# B&R Automation Studio project Parker_BMM_ST_V5_3147_V12 (part 30)

#### h_pid.c - Implementation code
```c
/********************************************************************
 * COPYRIGHT --
 ********************************************************************
 * Program: h_pid
 * File: h_pid.c
 * Author: lijianjun
 * Created: February 27, 2013
 ********************************************************************
 * Implementation of program h_pid -- heating and cooling controller
 ********************************************************************/

#include <bur/plctypes.h>
#include <string.h>

#ifdef _DEFAULT_INCLUDES
#include <AsDefault.h>
#endif

#include "edge.h"               /*edge function    */

#define  S$MODE_OFF					0
#define  S$MODE_PID					1
#define  S$MODE_TUNE					2

#define	C_STEP_WAIT 		   	0
#define	C_STEP_SYNC_HEAT_WAIT 	10
#define	C_STEP_HEAT 		    	20
#define	C_STEP_FREE 				30
#define	C_STEP_FREE_END			40
#define	C_STEP_COOL					50
#define	C_STEP_COOL_END 			60
#define	C_STEP_TUNE_END			70
#define	C_STEP_ERROR				999

void _INIT h_pidINIT(void)
{
	/* TODO: Add code here */
	gT_Par.Status.idxBroken = 0;
	gT_Par.Status.idxHigh   = 0;
	gT_Par.Status.idxLow    = 0;
	gT_Par.Status.idxFreeze = 0;
	gT_Par.Status.idxSwitchoff = 0;
	gT_Par.Status.idxNotNormal = 0;

	tProtectCooling = 0.0;

	/* ----- get task cycle time ----- */
	RTInfo_Task.enable = 1;
	RTInfo(&RTInfo_Task);

	tTask = RTInfo_Task.cycle_time/1000.0/1000.0;		/*  from us ---> s  */

	/* ----- setting tuning default value ----- */
	for(ZoneIndex=0; ZoneIndex<MAX_IDX_ZONE; ZoneIndex++)
	{
		/* parameter for tune   */
		LcrTempSet[ZoneIndex].TuneSet.delta_T_sync_heat = 40.0; 	 	/* Parameter for the synchronization  */
		LcrTempSet[ZoneIndex].TuneSet.delta_dT_sync_heat = 0.1;		/* Parameter for the synchronization d(temp)/dt  */
		LcrTempSet[ZoneIndex].TuneSet.cnt_wait_heat = 100;     		/* Parameter for the synchronization second  */

		LcrTempSet[ZoneIndex].TuneSet.delta_T_heat = 20.0;         	/* Parameter for the heating tuning 20 du */
		LcrTempSet[ZoneIndex].TuneSet.dT_min_heat  = 0.0;      		/* d(temp)/dt, min  */
		LcrTempSet[ZoneIndex].TuneSet.dRatio_heat  = 0.9;      		/* Internal parameter for the heating tuning 0 < dRatio_heat < 1*/
		LcrTempSet[ZoneIndex].TuneSet.cnt_tp_heat  = 180;      		/* 180  second */

		LcrTempSet[ZoneIndex].TuneSet.delta_T_sync_free  = 10.0; 	/* default value  */
		LcrTempSet[ZoneIndex].TuneSet.delta_dT_sync_free = 0.05;		/* default value   */
		LcrTempSet[ZoneIndex].TuneSet.cnt_wait_free      = 300;  	/* default value  300 second */

		LcrTempSet[ZoneIndex].TuneSet.delta_T_free = 10.0;				/* default value  10 du */
		LcrTempSet[ZoneIndex].TuneSet.dT_min_free  = 0.0;				/* default value  */
		LcrTempSet[ZoneIndex].TuneSet.dRatio_free  = 0.9;				/* default value  */
		LcrTempSet[ZoneIndex].TuneSet.cnt_tp_free  = 300;				/* default value  300 second */

		LcrTempSet[ZoneIndex].TuneSet.delta_T_sync_cool  = 10.0;		/* default value  10 du */
		LcrTempSet[ZoneIndex].TuneSet.delta_dT_sync_cool = 0.1;		/* not default value = 0.05  */
		LcrTempSet[ZoneIndex].TuneSet.cnt_wait_cool      = 300;		/* default value  300 second */

		LcrTempSet[ZoneIndex].TuneSet.delta_T_cool = 10.0;				/* default value  10 du */
		LcrTempSet[ZoneIndex].TuneSet.dT_min_cool  = 0.0;				/* default value  */
		LcrTempSet[ZoneIndex].TuneSet.dRatio_cool  = 0.9;				/* default value  */
		LcrTempSet[ZoneIndex].TuneSet.cnt_tp_cool  = 300.0;			/* default value  300 second */

		LcrTempSet[ZoneIndex].TuneSet.delta_T_sync_stop = 50.0;     /* Parameter for secure enable of the cooling tuning */
		LcrTempSet[ZoneIndex].TuneSet.filter_base_T = 20.0;         /* average value filter */
		LcrTempSet[ZoneIndex].TuneSet.Temp_amb = 40.0;

		LcrTempSet[ZoneIndex].TuneSet.mode = LCRTEMPTune_MODE_EXP;

		/* Heating and cooling mode  */
		LcrTempSet[ZoneIndex].enable_cooling  = 0;
		LcrTempSet[ZoneIndex].disable_heating = 0;

		/* stable parameter for PID   */
		LcrTempSet[ZoneIndex].PIDSet.hyst   = 2.0;
		LcrTempSet[ZoneIndex].PIDSet.Kw     = 1.0;
		LcrTempSet[ZoneIndex].PIDSet.delay  = 10.0;
		LcrTempSet[ZoneIndex].PIDSet.Kfbk   = 1.0;

		/* get address  */
		LCRTempTune_Array[ZoneIndex].pSettings = &(LcrTempSet[ZoneIndex]);
		LCRTempPID_Array[ZoneIndex].pSettings  = &(LcrTempSet[ZoneIndex]);

		gT_Par.Ctl.OnOff[ZoneIndex] = 0;
		gT_Par.Ctl.TuneOnOff[ZoneIndex] = 0;
		gT_Par.Ctl.IsHeatingOnPlan  = 0;
		gT_Par.Ctl.PreOnOff[ZoneIndex]= 0;
		gT_Par.Ctl.IsPreHeatingPlan = 0;

		OutBuffer[ZoneIndex]= 0.0;
		cntTask[ZoneIndex]  = 0;

		gT_Par.Status.TuneOk[ZoneIndex] = 0;

		HeatAlarm.tTempLow[ZoneIndex] = 1000.0;
	}/* for(ZoneIndex=0; ZoneIndex<MAX_ZoneIndex_CONTRL_ZONES; ZoneIndex++) */

}

void _CYCLIC h_pidCYCLIC(void)
{
	int i;
	gMachineInfo.bLoweringFlag =	bLowering; //ipis0424

	if (EDGEPOS(bLowering_Hmi,bLowering_Hmi_Pos))
	{
		if (1== gMachineOut.ParisonPump || 1== gMachineOut.ExtrA_Enable || 1==gMachineOut.ExtrB_Enable || gMachineOut.ExtrC_Enable || 1== gMachineOut.ExtrV_Enable)
		{
			gImply.ExtruderEnable =1;
		}
		else
		{
			bLowering =1;
		}
	}

	if (0==gMachineOut.HeatPower) //ipis0815
	{
		bLowering_Hmi =0;
	}

	if (0==bLowering_Hmi)
	{
		bLowering =0;
	}

	/* -------------------------------------------------------------------------- */
	if(1 == gT_Par.Ctl.IsAlarmConfirm)
	{
		gT_Par.Ctl.IsAlarmConfirm = 0;

		/* 非自复位的报警复位  */
		memset(gT_Par.Status.TempFreeze,0,sizeof(gT_Par.Status.TempFreeze));
		memset(gT_Par.Status.TempSwitchOff,0,sizeof(gT_Par.Status.TempSwitchOff));
	}

	/* -------------------------------------------------------------------------- */
	gT_Par.Status.idxBroken = 0;
	gT_Par.Status.idxHigh   = 0;
	gT_Par.Status.idxLow    = 0;
	gT_Par.Status.idxFreeze = 0;
	gT_Par.Status.idxSwitchoff = 0;
	gT_Par.Status.idxNotNormal = 0;

	gT_Par.Status.bBroken = 0;
	gT_Par.Status.bHigh   = 0;
	gT_Par.Status.bLowInternal = 0;
	gT_Par.Status.bFreeze = 0;
	gT_Par.Status.bSwitchOff = 0;
	gT_Par.Status.bNotNormal = 0;

	/*============================================================================*/
	/* Check group switches                              						         */
	/*============================================================================*/
	//	if(0 == gMachineIn.HeatingPowerNormal)gT_Par.GrpSwh.OnOff[0] = 0;
	if(0 == gMachineOut.HeatPower) gT_Par.GrpSwh.OnOff[0] = 0;

	if(0 == gT_Par.GrpSwh.OnOff[0] && 0 == gT_Par.GrpSwh.PreOnOff[0])
	{
		gMachineInfo.IsHeat = 0;
	}
	else if(1 == gT_Par.GrpSwh.OnOff[0] && 0 == gT_Par.GrpSwh.PreOnOff[0])
	{
		gMachineInfo.IsHeat = 1;
	}
	else
	{
		gMachineInfo.IsHeat = 2;
	}

	grpMaxIndex = sizeof(gT_Par.GrpSwh.OnOff)/sizeof(gT_Par.GrpSwh.OnOff[0]);
	if(grpMaxIndex > MAX_IDX_TEMPGROUP)grpMaxIndex = MAX_IDX_TEMPGROUP;

	for(grp=0; grp<grpMaxIndex; grp++)
	{
		if(gT_Par.Par.ST_GrpPreHeating[grp] < 20)gT_Par.Par.ST_GrpPreHeating[grp]= 20;
		if(gT_Par.Par.tGrpPreHeating[grp] < 10.0)gT_Par.Par.tGrpPreHeating[grp]  = 10.0;	/* 10.0min  */

		/* Pre-heating plan control  */
		if(1 == gT_Par.Ctl.IsPreHeatingPlan  && 0 == gT_Par.GrpSwh.PreOnOff[grp])
		{
			gMachineOut.HeatPower =1; //ipis0220
			gT_Par.GrpSwh.PreOnOff[grp] = 1;
			gT_Par.GrpSwh.OnOff[grp]    = 1;
		}

		if(1 == gT_Par.Ctl.IsHeatingOffPlan && 1 == gT_Par.GrpSwh.OnOff[grp])
		{
			gT_Par.GrpSwh.PreOnOff[grp] = 0;
		}

		if(0==gMachineIn.PreHeatDI)   //ipis0226
		{
			gT_Par.GrpSwh.PreOnOff[grp] = 0;
		}

		/* heating plan control  */
		if(1 == gT_Par.Ctl.IsHeatingOnPlan  && (0 == gT_Par.GrpSwh.OnOff[grp] || 1 == gT_Par.GrpSwh.PreOnOff[grp]))
		{
			gMachineOut.HeatPower =1; //ipis0220
			gT_Par.GrpSwh.OnOff[grp] = 1;
			gT_Par.GrpSwh.PreOnOff[grp] = 0;
		}

		if(1 == gT_Par.Ctl.IsHeatingOffPlan && 1 == gT_Par.GrpSwh.OnOff[grp])
		{
			gT_Par.GrpSwh.OnOff[grp] = 0;
		}

		/* Switch on group heating if group is on from VIS and programme enabled	*/
		if (EDGEPOS(gT_Par.GrpSwh.OnOff[grp],grp_OnOffPos[grp]))
		{
			HeatSequence[grp] = MAX_IDX_CONTRL_ZONES;
		}

		/* Switch off group heating if group is off from VIS and programe disabled	*/
		if (EDGENEG(gT_Par.GrpSwh.OnOff[grp],grp_OnOffNeg[grp]))
		{
			HeatSequence[grp] = 0;
			for(ZoneIndex=0;ZoneIndex<MAX_IDX_CONTRL_ZONES;ZoneIndex++)
			{
				if (gT_Par.Fix.SynchGroup[ZoneIndex] == grp)/*if grp nr configed     */
				{
					gT_Par.Ctl.OnOff[ZoneIndex] = 0;
				}
			}
		}
		/* Switch off group pre heating on  */
		if (EDGEPOS(gT_Par.GrpSwh.PreOnOff[grp],grp_PrePos[grp]))
		{
			for(ZoneIndex=0;ZoneIndex<MAX_IDX_CONTRL_ZONES;ZoneIndex++)
			{
				if (gT_Par.Fix.SynchGroup[ZoneIndex] == grp)/*if grp nr configed     */
				{
					gT_Par.Ctl.PreOnOff[ZoneIndex] = 1;
				}
			}
		}

		/* Switch off group pre heating off  */
		if (EDGENEG(gT_Par.GrpSwh.PreOnOff[grp],grp_PreNeg[grp]) || 0==gMachineIn.PreHeatDI) //ipis0221
		{
			for(ZoneIndex=0;ZoneIndex<MAX_IDX_CONTRL_ZONES;ZoneIndex++)
			{
				if (gT_Par.Fix.SynchGroup[ZoneIndex] == grp)/*if grp nr configed     */
				{
					gT_Par.Ctl.PreOnOff[ZoneIndex] = 0;
				}
			}
		}
		/* Switch off group tuning on  */
		if (EDGEPOS(gT_Par.GrpSwh.TuneOnOff[grp],grp_TunePos[grp]))
		{
			for(ZoneIndex=0;ZoneIndex<MAX_IDX_CONTRL_ZONES;ZoneIndex++)
			{
				if (gT_Par.Fix.SynchGroup[ZoneIndex] == grp)/*if grp nr configed     */
				{
					gT_Par.Ctl.TuneOnOff[ZoneIndex] = 1;
				}
			}
		}

		/* Switch off group tuning off  */
		if (EDGENEG(gT_Par.GrpSwh.TuneOnOff[grp],grp_TuneNeg[grp]))
		{
			for(ZoneIndex=0;ZoneIndex<MAX_IDX_CONTRL_ZONES;ZoneIndex++)
			{
				if (gT_Par.Fix.SynchGroup[ZoneIndex] == grp)/*if grp nr configed     */
				{
					gT_Par.Ctl.TuneOnOff[ZoneIndex] = 0;
				}
			}
		}

		grp_OnOffPos[grp] = gT_Par.GrpSwh.OnOff[grp];
		grp_OnOffNeg[grp] = gT_Par.GrpSwh.OnOff[grp];
	}/* for(grp=0; grp<grpMaxIndex; grp++) */

	/* Heat Sequence,one by one heat zone on */
	grpAct = grpMaxIndex;
	for(grp=0; grp<grpMaxIndex; grp++)
	{
		if(HeatSequence[grp] > 0)
		{
			grpAct = grp;
			break;
		}
	}

	if( grpAct < grpMaxIndex)
	{
		if(HeatSequence[grpAct] > 0)
		{
			if (grpAct == gT_Par.Fix.SynchGroup[MAX_IDX_CONTRL_ZONES - HeatSequence[grpAct]])
			{
				gT_Par.Ctl.OnOff[MAX_IDX_CONTRL_ZONES - HeatSequence[grpAct]] = 1;
			}
			HeatSequence[grpAct]--;
		}
	}

	/* check temperature change time  */
	if(gT_Par.Fix.tCheck < 10.0 )gT_Par.Fix.tCheck = 10.0;  /* 10.0s  */
	if(gT_Par.Fix.tHeatNormal < 20.0) gT_Par.Fix.tHeatNormal = 20.0;  /*  20.0 s */
	if(gT_Par.Fix.AT_MAX < 240.0)gT_Par.Fix.AT_MAX = 240.0; /* 240.0  */
	if(gT_Par.Par.ST_Tune_Same < 100)gT_Par.Par.ST_Tune_Same = 180.0;  /* Tune temperature   */

	/*============================================================================*/
	/* actual input && gAlarm check; PID parameters initialization   			  */
	/*============================================================================*/
	gMachineInfo.IsOpt = 0;
	for(ZoneIndex=0; ZoneIndex<MAX_IDX_CONTRL_ZONES; ZoneIndex++)
	{
		/*---UP-----------------------------------------------------------*/
		//		//		if (TempUpLimit_HMI[ZoneIndex]<=gT_Par.Fix.AT_MAX)
		//		//		{
		//		//			TempUpLimit_HMI[ZoneIndex] = gT_Par.Par.ST_PID[ZoneIndex]+  gUserFix_new.TempUpRange;
		//		//		}
		//		//		else
		//		//		{
		//		//			TempUpLimit_HMI[ZoneIndex] =gT_Par.Fix.AT_MAX;
		//		//		}
		//		//ipis022
		//		TempUpLimit_HMI[ZoneIndex] = gT_Par.Par.ST_PID[ZoneIndex]+  gUserFix_new.TempUpRange;
		//		if (gT_Par.Par.AlaUpTol[ZoneIndex] < gT_Par.Par.ST_PID[ZoneIndex] )
		//		{
		//			gT_Par.Par.AlaUpTol[ZoneIndex]=TempUpLimit_HMI[ZoneIndex];
		//		}
		//		//		if (gT_Par.Par.AlaUpTol[ZoneIndex] > gT_Par.Par.ST_PID[ZoneIndex] )
		//		//		{
		//		//			gT_Par.Par.AlaUpTol[ZoneIndex]=TempUpLimit_HMI[ZoneIndex];
		//		//		}
		//
		//		if (gT_Par.Par.AlaUpTol[ZoneIndex]>=TempUpLimit_HMI[ZoneIndex])
		//		{
		//			gT_Par.Par.AlaUpTol[ZoneIndex]=TempUpLimit_HMI[ZoneIndex];
		//		}
		//ipis0218
		if (gT_Par.Par.AlaUpTol[ZoneIndex] > gUserFix_new.TempUpRange )
		{
			gT_Par.Par.AlaUpTol[ZoneIndex]=gUserFix_new.TempUpRange;
		}
		if (gT_Par.Par.AlaUpTol[ZoneIndex] < 0 )
		{
			gT_Par.Par.AlaUpTol[ZoneIndex]=0;
		}
		/*---Down-----------------------------------------------------------*/
		//		if (TempUpLimit_HMI[ZoneIndex]>=0)
		//		{
		//			TempDwnLimit_HMI[ZoneIndex] = gT_Par.Par.ST_PID[ZoneIndex]- gUserFix_new.TempDwnRange;
		//		}
		//		else
		//		{
		//			TempDwnLimit_HMI[ZoneIndex] =0;
		//		}
		//		if(gT_Par.Par.AlaDwnTol[ZoneIndex]>gT_Par.Par.ST_PID[ZoneIndex])
		//		{
		//			gT_Par.Par.AlaDwnTol[ZoneIndex] = TempDwnLimit_HMI[ZoneIndex];
		//		}
		//		if(gT_Par.Par.AlaDwnTol[ZoneIndex]<TempDwnLimit_HMI[ZoneIndex])
		//		{
		//			gT_Par.Par.AlaDwnTol[ZoneIndex] = TempDwnLimit_HMI[ZoneIndex];
		//		}
		//
		//		if(gT_Par.Par.AlaDwnTol[ZoneIndex]<0)
		//		{
		//			gT_Par.Par.AlaDwnTol[ZoneIndex] = 0;
		//		}

		//ipis0218
		if(gT_Par.Par.AlaDwnTol[ZoneIndex]>gUserFix_new.TempDwnRange)
		{
			gT_Par.Par.AlaDwnTol[ZoneIndex] = gUserFix_new.TempDwnRange;
		}
		if(gT_Par.Par.AlaDwnTol[ZoneIndex]<0)
		{
			gT_Par.Par.AlaDwnTol[ZoneIndex] = 0;
		}

		/*---UP Same-----------------------------------------------------------*/
		//		if (TempUpLimit_Same_HMI<gT_Par.Fix.AT_MAX)
		//		{
		//			TempUpLimit_Same_HMI = gT_Par.Par.ST_PID_Same+  gUserFix_new.TempUpRange;
		//		}
		//		else
		//		{
		//			TempUpLimit_Same_HMI =gT_Par.Fix.AT_MAX;
		//		}
		//		TempUpLimit_Same_HMI = gT_Par.Par.ST_PID_Same+  gUserFix_new.TempUpRange;
		//		if (gT_Par.Par.AlaUpTol_Same<gT_Par.Par.ST_PID_Same)
		//		{
		//			gT_Par.Par.AlaUpTol_Same = TempUpLimit_Same_HMI;
		//		}
		//		//		if (gT_Par.Par.AlaUpTol_Same>gT_Par.Par.ST_PID_Same)
		//		//		{
		//		//			gT_Par.Par.AlaUpTol_Same = TempUpLimit_Same_HMI;
		//		//		}
		//		if (gT_Par.Par.AlaUpTol_Same>=TempUpLimit_Same_HMI)
		//		{
		//			gT_Par.Par.AlaUpTol_Same=TempUpLimit_Same_HMI;

		//ipis0218
		if (gT_Par.Par.AlaUpTol_Same > gUserFix_new.TempUpRange )
		{
			gT_Par.Par.AlaUpTol_Same=gUserFix_new.TempUpRange;
		}
		if (gT_Par.Par.AlaUpTol_Same < 0 )
		{
			gT_Par.Par.AlaUpTol_Same=0;
		}

		/*---Down Same-----------------------------------------------------------*/
		//		if (TempDwnLimit_Same_HMI>=0)
		//		{
		//			TempDwnLimit_Same_HMI = gT_Par.Par.ST_PID_Same- gUserFix_new.TempDwnRange;
		//		}
		//		else
		//		{
		//			TempDwnLimit_Same_HMI = 0;
		//		}
		//
		//		if (gT_Par.Par.AlaDwnTol_Same >gT_Par.Par.ST_PID_Same )
		//		{
		//			gT_Par.Par.AlaDwnTol_Same = TempDwnLimit_Same_HMI;
		//		}
		//		if (gT_Par.Par.AlaDwnTol_Same <TempDwnLimit_Same_HMI )
		//		{
		//			gT_Par.Par.AlaDwnTol_Same = TempDwnLimit_Same_HMI;
		//		}
		//		if (gT_Par.Par.AlaDwnTol_Same <0)
		//		{
		//			gT_Par.Par.AlaDwnTol_Same =0;
		//		}

		//ipis0218
		if(gT_Par.Par.AlaDwnTol_Same>gUserFix_new.TempDwnRange)
		{
			gT_Par.Par.AlaDwnTol_Same = gUserFix_new.TempDwnRange;
		}
		if(gT_Par.Par.AlaDwnTol_Same<0)
		{
			gT_Par.Par.AlaDwnTol_Same= 0;
		}

		//		TempUpLimit_HMI[ZoneIndex] = gT_Par.Par.ST_PID[ZoneIndex]+  gUserFix_new.TempUpRange;
		//
		//		TempDwnLimit_HMI[ZoneIndex] = gT_Par.Par.ST_PID[ZoneIndex]- gUserFix_new.TempDwnRange;
		//
		//		TempUpLimit_Same_HMI = gT_Par.Par.ST_PID_Same+  gUserFix_new.TempUpRange;
		//
		//		TempDwnLimit_Same_HMI = gT_Par.Par.ST_PID_Same- gUserFix_new.TempDwnRange;

		/*--------------------------------------------------------------*/

		gT_Par.Fix.bContactor[ZoneIndex] = 1;
		if(gT_Par.Fix.tTempFreeze[ZoneIndex] < 10.0 )gT_Par.Fix.tTempFreeze[ZoneIndex] = 10.0;
		if(gT_Par.Fix.tTempFreeze[ZoneIndex] > 1800.0)gT_Par.Fix.tTempFreeze[ZoneIndex] = 1800.0;

		if(tTask > 0.0 && 1 == gT_Par.Fix.Cooling[ZoneIndex])
		{
			gT_Par.Fix.tPeriodHeat[ZoneIndex] = ((INT)(gT_Par.Fix.tPeriodHeat[ZoneIndex]/tTask + 0.5)) * tTask;
			if(gT_Par.Fix.tPeriodHeat[ZoneIndex] < 10 * tTask)gT_Par.Fix.tPeriodHeat[ZoneIndex] = 10 * tTask;
		}

		if(tTask > 0.0 && 1 == gT_Par.Fix.bContactor[ZoneIndex])
		{
			gT_Par.Fix.tPeriodHeat[ZoneIndex] = ((INT)(gT_Par.Fix.tPeriodHeat[ZoneIndex]/tTask + 0.5)) * tTask;
			if(gT_Par.Fix.tPeriodHeat[ZoneIndex] < 10 * tTask)gT_Par.Fix.tPeriodHeat[ZoneIndex] = 10 * tTask;
		}

		/* ------ PID OPT value change ------ */
		if (memcmp(&gT_Par.Fix.ParTune[ZoneIndex],&ParTuneOld[ZoneIndex],sizeof(ParTuneOld[ZoneIndex])) != 0)
		{
			LcrTempSet[ZoneIndex].PIDpara = gT_Par.Fix.ParTune[ZoneIndex];
			LCRTempPID_Array[ZoneIndex].update = 1;
			ParTuneOld[ZoneIndex] = gT_Par.Fix.ParTune[ZoneIndex];
		}

		/* ---------------------- heating  normal -----------------------*/
		//ByPass gH_IO.HeatNormal(Feedback signal)which for detect heater error
		gH_IO.HeatNormal[ZoneIndex] = gH_IO.do_H[ZoneIndex];

		if(1 == gH_IO.do_H[ZoneIndex] && 0 == gH_IO.HeatNormal[ZoneIndex])
		{
			if(tHeatNormal[ZoneIndex] > 0.0)tHeatNormal[ZoneIndex] = tHeatNormal[ZoneIndex] - tTask;
			if(tHeatNormal[ZoneIndex] <= 0.0)
			{
				gT_Par.Status.bAlarmHeatNormal[ZoneIndex] = 1;
			}
		}
		else if(0 == gH_IO.do_H[ZoneIndex] && 1 == gH_IO.HeatNormal[ZoneIndex])
		{
			if(tHeatNormal[ZoneIndex] > 0.0)tHeatNormal[ZoneIndex] = tHeatNormal[ZoneIndex] - tTask;
			if(tHeatNormal[ZoneIndex] <= 0.0)
			{
				gT_Par.Status.bAlarmHeatNormal[ZoneIndex] = 1;
			}
		}
		else
		{
			gT_Par.Status.bAlarmHeatNormal[ZoneIndex] = 0;
			tHeatNormal[ZoneIndex] = gT_Par.Fix.tHeatNormal;
		}

		////ipis0719/////////////////////////////////////////////////////////////////////////////////////////////////////////////
		//		if (   0==TempInitOK[ZoneIndex]  )
		//		{
		//			//ipis0218
		//			if (( gH_IO.ActT[ZoneIndex] < gT_Par.Par.ST_PID[ZoneIndex] - gT_Par.Par.AlaDwnTol[ZoneIndex])&& 1 == gT_Par.Fix.Enable[ZoneIndex]
		//				|| 0==gMachineInfo.ExtrHeatTimeFlag) //ipis0213
		//			{
		//				gExtruderTempLow_HMIFlag =1;
		//			}
		//			else
		//			{
		//				gExtruderTempLow_HMIFlag =0;
		//			}
		//
		//		}

		/////////////////////////////////////////////////////////////////////////////////////////////////////////////////

		/* --- if current zone disabled, clear control bit --- */
		if (0 == gT_Par.Fix.Enable[ZoneIndex])
		{
			gT_Par.Ctl.OnOff[ZoneIndex] = 0;
			gT_Par.Ctl.TuneOnOff[ZoneIndex] = 0;

			gT_Par.Status.AlmHigh[ZoneIndex]      = 0;
			gT_Par.Status.AlmLow[ZoneIndex]       = 0;
			gT_Par.Status.SensorBroken[ZoneIndex] = 0;     /*For error bit show*/

			HeatAlarm.tSensorBroken[ZoneIndex] = 0.0;
			HeatAlarm.tTempHigh[ZoneIndex] = 0.0;
			HeatAlarm.tTempLow[ZoneIndex]  = 0.0;
			TempInitOK[ZoneIndex]=1;  //ipis0719

			//Bypass for gExtruderTempLow_HMIFlag
			TempProtection[ZoneIndex] =1;
			TempNotLow[ZoneIndex] =1;

		}
		else
		{
			if (1==gMachineInfo.IsHeat)
			{
				//	if (gH_IO.ActT[ZoneIndex] >= gT_Par.Par.AlaDwnTol[ZoneIndex])
				//ipis0218
				if (gH_IO.ActT[ZoneIndex] >= gT_Par.Par.ST_PID[ZoneIndex] - gT_Par.Par.AlaDwnTol[ZoneIndex])
				{
					{
						TempInitOK[ZoneIndex]=1;
					}

				}
				else
				{
					TempInitOK[ZoneIndex]=0;
				}

				if (1 == gT_Par.GrpSwh.OnOff[0])  //ipis 0128
				{
					gT_Par.Ctl.OnOff[ZoneIndex] = 1;
				}
				/*============================================================================*/
				/* Check gAlarm bit                                 						     */
				/*============================================================================*/
				/*-----------sensor broken or Opencircuit check-----------------------------*/
				if (gH_IO.ActT[ZoneIndex] >= 3000.0 || gH_IO.ActT[ZoneIndex] <= -3000.0)
				{
					HeatAlarm.tSensorBroken[ZoneIndex] = HeatAlarm.tSensorBroken[ZoneIndex] + tTask;

					if(HeatAlarm.tSensorBroken[ZoneIndex] > gT_Par.Fix.tCheck)
					{
						gT_Par.Status.SensorBroken[ZoneIndex] = 1;
					}
					else
					{
						gT_Par.Status.SensorBroken[ZoneIndex] = 0;
					}

					gT_Par.Status.AlmHigh[ZoneIndex] = 0;
					gT_Par.Status.AlmLow[ZoneIndex]  = 0;
					gT_Par.Status.TempFreeze[ZoneIndex] = 0;
				}
				else
				{
					HeatAlarm.tSensorBroken[ZoneIndex] = 0.0;
					gT_Par.Status.SensorBroken[ZoneIndex] = 0;

					if (1==gMachineInfo.IsHeat && (uDisHeaterTime>= gUserFix_new.HeatLowTimeOut*60))
					{
						//	if (gH_IO.ActT[ZoneIndex] < gT_Par.Par.AlaDwnTol[ZoneIndex])
						//ipis0218
						if (gH_IO.ActT[ZoneIndex] < gT_Par.Par.ST_PID[ZoneIndex]- gT_Par.Par.AlaDwnTol[ZoneIndex])
						{
							gAlarm.HeatError=1;
						}

					}

					if(1==TempInitOK[ZoneIndex] && 0== bLowering && 0==gT_Par.Ctl.IsPreHeatingPlan ) //ipis0304
					{
						/*Actual temperature high temp limit or upper tolerance limit*/
						//	if (gH_IO.ActT[ZoneIndex] > (gT_Par.Par.AlaUpTol[ZoneIndex]))/*Albert*/
						//ipis0211
						if (gH_IO.ActT[ZoneIndex] > (gT_Par.Par.ST_PID[ZoneIndex] +gT_Par.Par.AlaUpTol[ZoneIndex]))/*Albert*/
						{
							HeatAlarm.tTempHigh[ZoneIndex] = HeatAlarm.tTempHigh[ZoneIndex] + tTask;
							if(HeatAlarm.tTempHigh[ZoneIndex] > gT_Par.Fix.tCheck)
							{
								gT_Par.Status.AlmHigh[ZoneIndex] = 1;
							}
							else
							{
								gT_Par.Status.AlmHigh[ZoneIndex] = 0;
							}
						}
						else
						{
							HeatAlarm.tTempHigh[ZoneIndex] = 0.0;
							gT_Par.Status.AlmHigh[ZoneIndex] = 0;
						}

						/*Actual temperature low temp. limit or down tolerance limit*/
						//	if (gH_IO.ActT[ZoneIndex] < gT_Par.Par.AlaDwnTol[ZoneIndex])
						//ipis0218
						if (gH_IO.ActT[ZoneIndex] < gT_Par.Par.ST_PID[ZoneIndex] - gT_Par.Par.AlaDwnTol[ZoneIndex])

						{
							HeatAlarm.tTempLow[ZoneIndex] = HeatAlarm.tTempLow[ZoneIndex] + tTask;
							if(HeatAlarm.tTempLow[ZoneIndex] > gT_Par.Fix.tCheck)
							{
								gT_Par.Status.AlmLow[ZoneIndex] = 1;
							}
							else
							{
								gT_Par.Status.AlmLow[ZoneIndex] = 0;
							}
						}
						else
						{
							HeatAlarm.tTempLow[ZoneIndex] = 0.0;
							gT_Par.Status.AlmLow[ZoneIndex] = 0;
						}

						/*Actual temperature > permit max ---> stop heating */
						if ((gH_IO.ActT[ZoneIndex] > gT_Par.Fix.AT_MAX || gH_IO.ActT[ZoneIndex] < -100) &&
							(1 == gT_Par.Ctl.TuneOnOff[ZoneIndex] || 1 == gT_Par.Ctl.OnOff[ZoneIndex] || 1 == gT_Par.Ctl.PreOnOff[ZoneIndex])
							)
						{
							HeatAlarm.tTempSwitchOff[ZoneIndex] = HeatAlarm.tTempSwitchOff[ZoneIndex] + tTask;

							if(HeatAlarm.tTempSwitchOff[ZoneIndex] > gT_Par.Fix.tCheck)
							{
								gT_Par.Ctl.TuneOnOff[ZoneIndex] = 0;
								gT_Par.Ctl.OnOff[ZoneIndex]     = 0;
								gT_Par.Ctl.PreOnOff[ZoneIndex]  = 0;

								gT_Par.Status.TempSwitchOff[ZoneIndex] = 1;
							}
							else
							{
								gT_Par.Status.TempSwitchOff[ZoneIndex] = 0;
							}
						}
						else
						{
							HeatAlarm.tTempSwitchOff[ZoneIndex] = 0.0;
							gT_Par.Status.TempSwitchOff[ZoneIndex] = 0;

						}

					}
					else
					{
						gT_Par.Status.AlmHigh[ZoneIndex] = 0;
						gT_Par.Status.AlmLow[ZoneIndex] = 0;
						gT_Par.Status.TempSwitchOff[ZoneIndex] = 0;

					}

				}

			}

			//for gExtruderTempLow_HMIFlag
			if (gH_IO.ActT[ZoneIndex] > gUserFix_new.ProtectionTemp ) //ipis0225
			{
				TempProtection[ZoneIndex] =1;
			}
			else
			{
				TempProtection[ZoneIndex] =0;
			}

			if (gH_IO.ActT[ZoneIndex] < gT_Par.Par.ST_PID[ZoneIndex] - gT_Par.Par.AlaDwnTol[ZoneIndex] ) //0226
			{
				TempNotLow[ZoneIndex] =0;
			}
			else
			{
				TempNotLow[ZoneIndex] =1;
			}

		}/* if (0 == gT_Par.Fix.Enable[ZoneIndex]) */

		/* PID and TUNE get set parameter address  */
		LCRTempPID_Array[ZoneIndex].pSettings  = &LcrTempSet[ZoneIndex];
		LCRTempTune_Array[ZoneIndex].pSettings = &LcrTempSet[ZoneIndex];

		/* act temperature */
		LCRTempPID_Array[ZoneIndex].Temp  = gH_IO.ActT[ZoneIndex];
		LCRTempTune_Array[ZoneIndex].Temp = gH_IO.ActT[ZoneIndex];

		/*  set temperature */
		if(1 == gT_Par.Ctl.PreOnOff[ZoneIndex])
		{
			for(grp=0; grp<grpMaxIndex; grp++)
			{
				if (gT_Par.Fix.SynchGroup[ZoneIndex] == grp)
				{
					LCRTempPID_Array[ZoneIndex].Temp_set = gT_Par.Par.ST_GrpPreHeating[grp];
				}
			}
		}
		else
		{
			/*2018.7.31 Albert add new lowering setting*/
			//			LCRTempPID_Array[ZoneIndex].Temp_set = gT_Par.Par.ST_PID[ZoneIndex];
			if(1 == bLowering)	LCRTempPID_Array[ZoneIndex].Temp_set = gT_Par.Par.ST_PID[ZoneIndex] - gT_Par.Par.Lower;
			else LCRTempPID_Array[ZoneIndex].Temp_set = gT_Par.Par.ST_PID[ZoneIndex];

		}

		gT_Par.Par.ST_Tune[ZoneIndex] = gT_Par.Par.ST_Tune_Same;
		LCRTempTune_Array[ZoneIndex].Temp_set = gT_Par.Par.ST_Tune[ZoneIndex];

		//		/* Preheating on time --> Preheating off, normal heating*/
		//		if(1 == gT_Par.Ctl.PreOnOff[ZoneIndex])
		//		{
		//			/* reach setting pre-heating temperature - 5.0 */
		//			if( gH_IO.ActT[ZoneIndex] > LCRTempPID_Array[ZoneIndex].Temp_set - 5.0)
		//			{
		//				HeatTest.tPreHeating[ZoneIndex] = HeatTest.tPreHeating[ZoneIndex] + tTask;
		//			}
		//			else
		//			{
		//				HeatTest.tPreHeating[ZoneIndex] = 0.0;
		//			}
		//
		//			for(grp=0; grp<grpMaxIndex; grp++)
		//			{
		//				if (gT_Par.Fix.SynchGroup[ZoneIndex] == grp)
		//				{
		//					if(HeatTest.tPreHeating[ZoneIndex] > gT_Par.Par.tGrpPreHeating[grp] * 60)
		//					{
		//						gT_Par.Ctl.OnOff[ZoneIndex]    = 1;
		//						gT_Par.Ctl.PreOnOff[ZoneIndex] = 0;
		//						gT_Par.Status.PreHeatingOk[ZoneIndex] = 1;
		//					}
		//				}
		//			}
		//		}
		//		else
		//		{
		//			HeatTest.tPreHeating[ZoneIndex] = 0;
		//		}

		/* Heating Power not Normal, single zone not permit heating  */
		if(0 == gMachineIn.HeatingPowerNormal)
		{
			gT_Par.Ctl.OnOff[ZoneIndex] = 0;
			gT_Par.Ctl.PreOnOff[ZoneIndex] = 0;
		}

		/* off or PID or tuning  */
		if ((1 == gT_Par.Status.SensorBroken[ZoneIndex]) || (0 == gT_Par.Fix.Enable[ZoneIndex]))     /*sensor broken*/
		{
			PIDSTEP[ZoneIndex] = S$MODE_OFF;			/* If sensor error or not anble --> switch off zone		*/

			gT_Par.Ctl.OnOff[ZoneIndex]     = 0;
			gT_Par.Ctl.TuneOnOff[ZoneIndex] = 0;
			gT_Par.Ctl.PreOnOff[ZoneIndex]  = 0;

			gT_Par.Status.Tuning[ZoneIndex] = 0;
			gT_Par.Status.TuneStatus[ZoneIndex] = 0;
		}
		else if ((1 == gT_Par.Ctl.TuneOnOff[ZoneIndex]) && (1 == gT_Par.Ctl.OnOff[ZoneIndex]))
		{
			PIDSTEP[ZoneIndex] = S$MODE_TUNE;		/* Tune mode*/

			gT_Par.Status.Tuning[ZoneIndex] = 1;
			gMachineInfo.IsOpt  =  1;
		}
		else if ((1 == gT_Par.Ctl.OnOff[ZoneIndex]) || (1 == gT_Par.Ctl.PreOnOff[ZoneIndex]))
		{
			PIDSTEP[ZoneIndex] = S$MODE_PID;			/* PID mode*/

			gT_Par.Status.Tuning[ZoneIndex] = 0;
			gT_Par.Status.TuneStatus[ZoneIndex] = 0;
		}
		else
		{
			PIDSTEP[ZoneIndex] = S$MODE_OFF;

			gT_Par.Ctl.OnOff[ZoneIndex]     = 0;
			gT_Par.Status.Tuning[ZoneIndex] = 0;
		}

		/* step machine for temperature control  */
		switch (PIDSTEP[ZoneIndex])
		{
			case S$MODE_OFF:
					LcrTempSet[ZoneIndex].enable_cooling = 0;

				gH_IO.y_heat[ZoneIndex] = 0;
				gH_IO.y_cool[ZoneIndex] = 0;

				cntTask[ZoneIndex] = 0;
				OutBuffer[ZoneIndex] = 0.0;

				HeatTest.tTempFreeze[ZoneIndex] = 0.0;
				gT_Par.Status.PreHeatingOk[ZoneIndex] = 0;

				StepTune[ZoneIndex] = C_STEP_WAIT;

				LCRTempTune_Array[ZoneIndex].okToCool    = 0;
				LCRTempTune_Array[ZoneIndex].okToCoolEnd = 0;
				LCRTempTune_Array[ZoneIndex].okToFree    = 0;
				LCRTempTune_Array[ZoneIndex].okToFreeEnd = 0;
				LCRTempTune_Array[ZoneIndex].okToHeat    = 0;

				LCRTempPID_Array[ZoneIndex].enable  = 0;
				LCRTempTune_Array[ZoneIndex].enable = 0;

				gT_Par.Status.Out[ZoneIndex] = 0.0;
				break;

			case S$MODE_PID:
					LCRTempPID_Array[ZoneIndex].enable  = 1;
				LCRTempTune_Array[ZoneIndex].enable = 0;

				StepTune[ZoneIndex] = C_STEP_WAIT;

				LCRTempPID_Array[ZoneIndex].mode = LCRTEMPPID_MODE_AUTO;

				LcrTempSet[ZoneIndex].PIDpara = gT_Par.Fix.ParTune[ZoneIndex];

				/* heating default setting pid parameter  */
				if(0.0 == LcrTempSet[ZoneIndex].PIDpara.Kp_h)LcrTempSet[ZoneIndex].PIDpara.Kp_h = 3.0;
				if(0.0 == LcrTempSet[ZoneIndex].PIDpara.Tn_h)LcrTempSet[ZoneIndex].PIDpara.Tn_h = 5.0;
				if(0.0 == LcrTempSet[ZoneIndex].PIDpara.Tv_h)LcrTempSet[ZoneIndex].PIDpara.Tv_h = 1.0;

				/* ------ option cooling ------ */
				if(LcrTempSet[ZoneIndex].enable_cooling != gT_Par.Fix.Cooling[ZoneIndex])
				{
					LCRTempPID_Array[ZoneIndex].update = 1;
					LcrTempSet[ZoneIndex].enable_cooling = gT_Par.Fix.Cooling[ZoneIndex];
				}

				/* cooling default setting pid parameter  */
				if(LcrTempSet[ZoneIndex].PIDpara.Kp_c < 0.1)LcrTempSet[ZoneIndex].PIDpara.Kp_c = 6.0;
				LcrTempSet[ZoneIndex].PIDpara.Tn_c = 0.0;
				LcrTempSet[ZoneIndex].PIDpara.Tv_c = 0.0;
				if(0 == ZoneIndex)LcrTempSet[ZoneIndex].PIDpara.Kp_c = 5.0;
				/* Calling fuction LCRTempPID  */
				LCRTempPID(&LCRTempPID_Array[ZoneIndex]);

				if(0 == LcrTempSet[ZoneIndex].enable_cooling && 0 == gT_Par.Fix.bContactor[ZoneIndex])	/*  only heating && not contactor heating*/
				{
					gH_IO.y_heat[ZoneIndex] = LCRTempPID_Array[ZoneIndex].y_heat;
					gH_IO.y_cool[ZoneIndex] = LCRTempPID_Array[ZoneIndex].y_cool;
				}
				else   /* heating and cooling */
				{
					cntSamples[ZoneIndex] = (UINT)(gT_Par.Fix.tPeriodHeat[ZoneIndex]/tTask + 0.1);
					if(cntSamples[ZoneIndex] > 0)
					{
						if(0 == (cntTask[ZoneIndex] % cntSamples[ZoneIndex]))
						{
							OutBuffer[ZoneIndex] = OutBuffer[ZoneIndex] + (LCRTempPID_Array[ZoneIndex].y_heat - LCRTempPID_Array[ZoneIndex].y_cool)/cntSamples[ZoneIndex];
							if(OutBuffer[ZoneIndex] >= 100.0)
							{
								OutBuffer[ZoneIndex] = OutBuffer[ZoneIndex] - 100.0;
								gH_IO.y_heat[ZoneIndex] = 100.0;
								gH_IO.y_cool[ZoneIndex] = 0.0;
							}
							else if(OutBuffer[ZoneIndex] <= -100.0)
							{
								OutBuffer[ZoneIndex] = OutBuffer[ZoneIndex] + 100.0;
								gH_IO.y_heat[ZoneIndex] = 0.0;
								gH_IO.y_cool[ZoneIndex] = 100;
							}
							else
							{
								gH_IO.y_heat[ZoneIndex] = 0.0;
								gH_IO.y_cool[ZoneIndex] = 0.0;
							}
						}
						else
						{
							OutBuffer[ZoneIndex] = OutBuffer[ZoneIndex] + (LCRTempPID_Array[ZoneIndex].y_heat - LCRTempPID_Array[ZoneIndex].y_cool)/cntSamples[ZoneIndex];
						}
					}
					else
					{
						gH_IO.y_heat[ZoneIndex] = LCRTempPID_Array[ZoneIndex].y_heat;
						gH_IO.y_cool[ZoneIndex] = LCRTempPID_Array[ZoneIndex].y_cool;
					}
				}

				cntTask[ZoneIndex] = cntTask[ZoneIndex] ++;
				if(cntTask[ZoneIndex]>= 10000)cntTask[ZoneIndex]= 1000;

				/* zone output percent  */
				if(LCRTempPID_Array[ZoneIndex].y_heat > 0)
				{
					gT_Par.Status.Out[ZoneIndex] = LCRTempPID_Array[ZoneIndex].y_heat;
				}
				else if (LCRTempPID_Array[ZoneIndex].y_cool > 0)
				{
					gT_Par.Status.Out[ZoneIndex] = - LCRTempPID_Array[ZoneIndex].y_cool;
				}
				else
				{
					gT_Par.Status.Out[ZoneIndex] = 0.0;
				}

				/* Heating excption -- sensor   */
				if(100.0 == LCRTempPID_Array[ZoneIndex].y_heat)
				{
					HeatTest.tTempFreeze[ZoneIndex] = HeatTest.tTempFreeze[ZoneIndex] +  tTask;
				}
				else
				{
					HeatTest.tTempFreeze[ZoneIndex] = 0.0;
				}

				if(tTask * 2 == HeatTest.tTempFreeze[ZoneIndex])
				{
					HeatTest.LastTemp[ZoneIndex] = LCRTempPID_Array[ZoneIndex].Temp;
				}

				if(gT_Par.Fix.tTempFreeze[ZoneIndex] == HeatTest.tTempFreeze[ZoneIndex] + tTask * 2)
				{
					if(LCRTempPID_Array[ZoneIndex].Temp < HeatTest.LastTemp[ZoneIndex] + 1.0)
					{
						gT_Par.Status.TempFreeze[ZoneIndex] = 1;
						if(1 == gT_Par.Fix.ProtectEna[ZoneIndex])
						{
							gT_Par.Ctl.OnOff[ZoneIndex]    = 0;
							gT_Par.Ctl.PreOnOff[ZoneIndex] = 0;
						}
					}
				}
				break;

			case S$MODE_TUNE:
					LCRTempPID_Array[ZoneIndex].enable  = 0;
				LCRTempTune_Array[ZoneIndex].enable = 1;

				/* ------ option cooling ------ */
				if(LcrTempSet[ZoneIndex].enable_cooling != 0)
				{
					LCRTempPID_Array[ZoneIndex].update = 1;
					LcrTempSet[ZoneIndex].enable_cooling = 0;
				}

				cntTask[ZoneIndex] = 0;
				OutBuffer[ZoneIndex] = 0.0;

				/* tuning step machine   */
				switch (StepTune[ZoneIndex])
				{
					/* ------- step start ------- */
					case C_STEP_WAIT:
						if(1 == gT_Par.Ctl.TuneOnOff[ZoneIndex])
						{
							gT_Par.Status.TuneOk[ZoneIndex] = 0;
							LCRTempTune_Array[ZoneIndex].start = 1;
							StepTune[ZoneIndex] = C_STEP_SYNC_HEAT_WAIT;
						}
						break;

					/* ------- step sync heat ------- */
					case C_STEP_SYNC_HEAT_WAIT:

						LCRTempTune_Array[ZoneIndex].okToHeat = 1;

						for( i=0; i<MAX_IDX_CONTRL_ZONES;i++)
						{
							if(1 == gT_Par.Ctl.TuneOnOff[i])
							{
								gT_Par.Status.okToHeat[i] = LCRTempTune_Array[i].rdyToHeat;
							}
							else
							{
								gT_Par.Status.okToHeat[i] = 1;
							}

							LCRTempTune_Array[ZoneIndex].okToHeat = LCRTempTune_Array[ZoneIndex].okToHeat & gT_Par.Status.okToHeat[i];
						}

						if(1 == LCRTempTune_Array[ZoneIndex].okToHeat)
						{
							StepTune[ZoneIndex] = C_STEP_HEAT;
						}
						break;

					/* ------- step  heating ------- */
					case C_STEP_HEAT:

						LCRTempTune_Array[ZoneIndex].okToFree = 1;

						for( i=0; i<MAX_IDX_CONTRL_ZONES;i++)
						{
							if(1 == gT_Par.Ctl.TuneOnOff[i])
							{
								gT_Par.Status.okToFree[i] = LCRTempTune_Array[i].rdyToFree;
							}
							else
							{
								gT_Par.Status.okToFree[i] = 1;
							}

							LCRTempTune_Array[ZoneIndex].okToFree = LCRTempTune_Array[ZoneIndex].okToFree & gT_Par.Status.okToFree[i];
						}

						if(1 == LCRTempTune_Array[ZoneIndex].okToFree)
						{
							StepTune[ZoneIndex] = C_STEP_FREE;
						}
						break;

					/* ------- step  heating free ------- */
					case  C_STEP_FREE:

						LCRTempTune_Array[ZoneIndex].okToFreeEnd = 1;

						for( i=0; i<MAX_IDX_CONTRL_ZONES;i++)
						{
							if(1 == gT_Par.Ctl.TuneOnOff[i])
							{
								gT_Par.Status.okToFreeEnd[i] = LCRTempTune_Array[i].rdyToFreeEnd;
							}
							else
							{
								gT_Par.Status.okToFreeEnd[i] = 1;
							}

							LCRTempTune_Array[ZoneIndex].okToFreeEnd = LCRTempTune_Array[ZoneIndex].okToFreeEnd & gT_Par.Status.okToFreeEnd[i];
						}

						if(1 == LCRTempTune_Array[ZoneIndex].okToFreeEnd)
						{
							StepTune[ZoneIndex] = C_STEP_FREE_END;
						}
						break;

					/* ------- step  heating free end ------- */
					case C_STEP_FREE_END:

						LCRTempTune_Array[ZoneIndex].okToCool = 1;

						for( i=0; i<MAX_IDX_CONTRL_ZONES;i++)
						{
							if(1 == gT_Par.Ctl.TuneOnOff[i])
							{
								gT_Par.Status.okToCool[i] = LCRTempTune_Array[i].rdyToCool;
							}
							else
							{
								gT_Par.Status.okToCool[i] = 1;
							}

							LCRTempTune_Array[ZoneIndex].okToCool = LCRTempTune_Array[ZoneIndex].okToCool & gT_Par.Status.okToCool[i];
						}

						if(1 == LCRTempTune_Array[ZoneIndex].okToCool)
						{
							StepTune[ZoneIndex] = C_STEP_COOL;
						}
						break;
					/* ------- step  cooling ------- */
					case C_STEP_COOL:

						LCRTempTune_Array[ZoneIndex].okToCoolEnd = 1;

						for( i=0; i<MAX_IDX_CONTRL_ZONES;i++)
						{
							if(1 == gT_Par.Ctl.TuneOnOff[i])
							{
								gT_Par.Status.okToCoolEnd[i] = LCRTempTune_Array[i].rdyToCoolEnd;
							}
							else
							{
								gT_Par.Status.okToCoolEnd[i] = 1;
							}

							LCRTempTune_Array[ZoneIndex].okToCoolEnd = LCRTempTune_Array[ZoneIndex].okToCoolEnd & gT_Par.Status.okToCoolEnd[i];
						}

						if(1 == LCRTempTune_Array[ZoneIndex].okToCoolEnd)
						{
							StepTune[ZoneIndex] = C_STEP_COOL_END;
						}
						break;

					/* ------- step  cooling end ------- */
					case C_STEP_COOL_END:
						if(1 == LCRTempTune_Array[ZoneIndex].done)
						{
							gT_Par.Status.TuneOk[ZoneIndex] = 1;
							StepTune[ZoneIndex] = C_STEP_TUNE_END;
						}
						break;

					/* ------- step  tune end ------- */
					case C_STEP_TUNE_END:
						LCRTempTune_Array[ZoneIndex].start = 0;
						gT_Par.Ctl.TuneOnOff[ZoneIndex] = 0;

						gT_Par.Fix.ParTune[ZoneIndex] = LcrTempSet[ZoneIndex].PIDpara;

						StepTune[ZoneIndex] = C_STEP_WAIT;
						break;

					/* ------- step  heating error ------- */
					case C_STEP_ERROR:
						gT_Par.Ctl.TuneOnOff[ZoneIndex] = 0;
						gT_Par.Ctl.OnOff[ZoneIndex]     = 0;
						gT_Par.Ctl.PreOnOff[ZoneIndex]  = 0;
						break;

				}/* switch (StepTune[ZoneIndex]) */

				/* Calling fuction LCRTempTune  */
				LCRTempTune(&LCRTempTune_Array[ZoneIndex]);

				if(LCRTempTune_Array[ZoneIndex].status >= LCR_ERR_LCRPIDTune_ABORT && LCRTempTune_Array[ZoneIndex].status <= LCR_ERR_LCRPIDTune_W_CHANGED)
				{
					StepTune[ZoneIndex] = C_STEP_ERROR;
				}

				gT_Par.Status.TuneStatus[ZoneIndex] = StepTune[ZoneIndex];

				gH_IO.y_heat[ZoneIndex] = LCRTempTune_Array[ZoneIndex].y_heat;
				gH_IO.y_cool[ZoneIndex] = LCRTempTune_Array[ZoneIndex].y_cool;

				/* zone output percent  */
				if(LCRTempTune_Array[ZoneIndex].y_heat > 0)
				{
					gT_Par.Status.Out[ZoneIndex] = LCRTempTune_Array[ZoneIndex].y_heat;
				}
				else if (LCRTempTune_Array[ZoneIndex].y_cool > 0)
				{
					gT_Par.Status.Out[ZoneIndex] = - LCRTempTune_Array[ZoneIndex].y_cool;
				}
				else
				{
					gT_Par.Status.Out[ZoneIndex] = 0.0;
				}

				if(100.0 == LCRTempTune_Array[ZoneIndex].y_heat)
				{
					HeatTest.tTempFreeze[ZoneIndex] = HeatTest.tTempFreeze[ZoneIndex] +  tTask;
				}
				else
				{
					HeatTest.tTempFreeze[ZoneIndex] = 0.0;
				}

				if(tTask * 2 == HeatTest.tTempFreeze[ZoneIndex])
				{
					HeatTest.LastTemp[ZoneIndex] = LCRTempPID_Array[ZoneIndex].Temp;
				}

				if(gT_Par.Fix.tTempFreeze[ZoneIndex] == HeatTest.tTempFreeze[ZoneIndex] + tTask * 2)
				{
					if(LCRTempPID_Array[ZoneIndex].Temp < HeatTest.LastTemp[ZoneIndex] + 1.0)
					{
						gT_Par.Status.TempFreeze[ZoneIndex] = 1;
						if(1 == gT_Par.Fix.ProtectEna[ZoneIndex])
						{
							gT_Par.Ctl.OnOff[ZoneIndex] = 0;
						}
					}
				}
				break;
		}/* switch (PIDSTEP[ZoneIndex]) */

		/* ------------------ gAlarm idex information ------------------ */
		if(1 == gT_Par.Status.SensorBroken[ZoneIndex])
		{
			gT_Par.Status.idxBroken = ZoneIndex + 1;
			gT_Par.Status.bBroken = 1;
		}

		if(1 == gT_Par.Status.AlmHigh[ZoneIndex])
		{
			gT_Par.Status.idxHigh = ZoneIndex + 1;
			gT_Par.Status.bHigh = 1;
		}

		if(1 == gT_Par.Status.AlmLow[ZoneIndex])
		{
			gT_Par.Status.idxLow = ZoneIndex + 1;
			gT_Par.Status.bLowInternal = 1;
		}

		if(1 == gT_Par.Status.TempSwitchOff[ZoneIndex])
		{
			gT_Par.Status.idxSwitchoff = ZoneIndex + 1;
			gT_Par.Status.bSwitchOff = 1;
		}

		if(1 == gT_Par.Status.TempFreeze[ZoneIndex])
		{
			gT_Par.Status.idxFreeze = ZoneIndex + 1;
			gT_Par.Status.bFreeze = 1;
		}

		if(1 == gT_Par.Status.bAlarmHeatNormal[ZoneIndex])
		{
			gT_Par.Status.bNotNormal = 1;
			gT_Par.Status.idxNotNormal = ZoneIndex + 1;
		}

		TempInitOK_Old[ZoneIndex] =1; //ipis0218

	}/* for(ZoneIndex=0; ZoneIndex<MAX_ZoneIndex_CONTRL_ZONES; ZoneIndex++) */
	////ipis0218
	gTempfirstHeatOK = memcmp(&TempInitOK, &TempInitOK_Old , sizeof(TempInitOK));//0= all OK
	TempProtectionFlag = memcmp(&TempProtection, &TempInitOK_Old , sizeof(TempProtection));  //0= all OK
	TempNotLowFlag = memcmp(&TempNotLow, &TempInitOK_Old , sizeof(TempNotLow)); //0= all OK

	if (0==gMachineInfo.IsHeat)
	{
		TempProtectionFix_HMI =1;
	}
	if (EDGEPOS(gMachineInfo.IsHeat,IsHeatPos))
	{
		if (0==TempProtectionFlag)
		{
			TempProtectionMode =1; //mold
			TempProtectionFix_HMI =1;
		}
		else
		{
			TempProtectionMode =0;	//fix
			TempProtectionFix_HMI =0;
		}
	}

	//	if (0==gTempfirstHeatOK) //ipis0225
	if (1==gMachineInfo.IsHeat && 0==gTempfirstHeatOK)
	{
		if (0==TempProtectionMode) //fix ipis0225
		{
			//			if (tProtectCooling < gT_Par.Fix.tProtectCoolingFix+10)
			//			{
			//				tProtectCooling = tProtectCooling + tTask;
			//			}
			//			if (tProtectCooling > gT_Par.Fix.tProtectCoolingFix ) //ipis0218 force first power on and first heat, must wait 20min
			//			{
			//				gMachineInfo.ExtrHeatTimeFlag =1;
			//					TempProtectionFix_HMI =1;
			//			}
			if (tProtectCooling < gT_Par.Fix.tProtectCoolingFix+10 || tProtectCooling < gT_Par.Fix.tProtectCooling+10)
			{
				tProtectCooling = tProtectCooling + tTask;
				if(tProtectCooling > gT_Par.Fix.tProtectCoolingFix)
				{
					TempProtectionFix_HMI =1;
				}
			}
			if (tProtectCooling > gT_Par.Fix.tProtectCoolingFix  && tProtectCooling > gT_Par.Fix.tProtectCooling ) //ipis0218 force first power on and first heat, must wait 20min
			{
				gMachineInfo.ExtrHeatTimeFlag =1;
				TempProtectionFix_HMI =1;
			}
		}
		else
		{
			if (tProtectCooling < gT_Par.Fix.tProtectCooling+10)
			{
				tProtectCooling = tProtectCooling + tTask;
			}
			if (tProtectCooling > gT_Par.Fix.tProtectCooling )
			{
				gMachineInfo.ExtrHeatTimeFlag =1;
			}
		}
	}
	else
	{
		tProtectCooling =0;
		gMachineInfo.ExtrHeatTimeFlag =0;
	}

	//ipis0226
	//gTempfirstHeatOK  =
	// TempNotLowFlag = all enable zone temp is in setting range
	// gMachineInfo.ExtrHeatTimeFlag  =
	if (0==gTempfirstHeatOK && 0== TempNotLowFlag && 1==gMachineInfo.ExtrHeatTimeFlag) //ipis0213
	{
		gExtruderTempLow_HMIFlag =0;
	}
	else
	{
		gExtruderTempLow_HMIFlag =1;
	}

	//ipis0213 	/* extruder protection cooling   */
	//	if (0==gTempfirstHeatOK)
	//	{
	//		tProtectCooling = tProtectCooling + tTask;
	//
	//
	//		if (1== gMachineInfo.ExtrHeatTimeFlag) //=ipis0225
	//		{
	//			if (tProtectCooling < gT_Par.Fix.tProtectCooling+10)
	//			{
	//				tProtectCooling = tProtectCooling + tTask;
	//			}
	//		}
	//		else
	//		{
	//			if (tProtectCooling < gT_Par.Fix.tProtectCoolingFix+10)
	//			{
	//				tProtectCooling = tProtectCooling + tTask;
	//			}
	//		}
	//
	//
	//		if (1== gMachineInfo.ExtrHeatTimeFlag)
	//		{
	//			if (tProtectCooling > gT_Par.Fix.tProtectCooling )
	//			{
	//				gMachineInfo.ExtrHeatTimeFlag =1;
	//			}
	//		}
	//		else
	//		{
	//			if (tProtectCooling > gT_Par.Fix.tProtectCoolingFix ) //ipis0218 force first power on and first heat, must wait 20min
	//			{
	//				gMachineInfo.ExtrHeatTimeFlag =1;
	//			}
	//
	//		}
	//
	//	}
	//	else
	//	{
	//		tProtectCooling =0;
	//		gMachineInfo.ExtrHeatTimeFlag =0;
	//	}

	/* extruder protection cooling   */
	if(0 == gT_Par.Status.bLowInternal)
	{
		//		tProtectCooling = tProtectCooling + tTask;
		//		if(tProtectCooling > 2 * gT_Par.Fix.tProtectCooling)
		//		{
		//			tProtectCooling = 2 * gT_Par.Fix.tProtectCooling + 1.0;
		//		}
		gT_Par.Status.bLow = 0;
		//		if(tProtectCooling >= gT_Par.Fix.tProtectCooling)
		//		{
		//			gT_Par.Status.bLow = 0;
		//		}
		//		else
		//		{
		//			gT_Par.Status.bLow = 1;
		//		}
	}
	else
	{
		//		tProtectCooling = 0.0;
		gT_Par.Status.bLow = 1;
		//	gT_Par.Status.bLow = 0; //ipis0227
	}

	/*2018.7.24 Albert add timer show heat time*/
	if(gMachineInfo.IsHeat && 0== bLowering)
	{
		rHeaterTime += tTask;
	}
	else
	{
		rHeaterTime = 0;
	}
	uDisHeaterTime = rHeaterTime;

}/* end of CYCLIC   */
```

#### h_pid.typ - Local data types
```iecst
(********************************************************************
 * COPYRIGHT --
 ********************************************************************
 * Program: h_pid
 * File: h_pid.typ
 * Author: lij
 * Created: February 27, 2013
 ********************************************************************
 * Local data types of program h_pid
 ********************************************************************)

TYPE
	Heat_Alarm_typ : 	STRUCT
		tTempSwitchOff : ARRAY[0..MAX_IDX_ZONE]OF REAL;
		tSensorBroken : ARRAY[0..MAX_IDX_ZONE]OF REAL;
		tTempHigh : ARRAY[0..MAX_IDX_ZONE]OF REAL;
		tTempLow : ARRAY[0..MAX_IDX_ZONE]OF REAL;
	END_STRUCT;
	Heat_Test_typ : 	STRUCT
		LastTemp : ARRAY[0..MAX_IDX_ZONE]OF REAL;
		tTempFreeze : ARRAY[0..MAX_IDX_ZONE]OF REAL;
		tPreHeating : ARRAY[0..MAX_IDX_ZONE]OF REAL;
	END_STRUCT;
END_TYPE
```

#### h_pid.var - Local variables
```iecst
(********************************************************************
 * COPYRIGHT --
 ********************************************************************
 * Program: h_pid
 * File: h_pid.var
 * Author: lij
 * Created: February 27, 2013
 ********************************************************************
 * Local variables of program h_pid
 ********************************************************************)
VAR
	ZoneIndex : UINT;
	tTask : REAL := 0.0;
	tProtectCooling : REAL;
	StepTune : ARRAY[0..MAX_IDX_ZONE] OF UINT;
	RTInfo_Task : RTInfo := (0);
	PIDSTEP : ARRAY[0..MAX_IDX_ZONE] OF UINT;
	ParTuneOld : ARRAY[0..MAX_IDX_ZONE] OF lcrtemp_pid_opt_typ;
	LCRTempTune_Array : ARRAY[0..MAX_IDX_ZONE] OF LCRTempTune := [MAX_IDX_ZONE+1(0)];
END_VAR
VAR RETAIN
	LcrTempSet : ARRAY[0..MAX_IDX_ZONE] OF lcrtemp_set_typ;
END_VAR
VAR
	LCRTempPID_Array : ARRAY[0..MAX_IDX_ZONE] OF LCRTempPID := [MAX_IDX_ZONE+1(0)];
	tHeatNormal : ARRAY[0..MAX_IDX_ZONE] OF REAL;
	OutBuffer : ARRAY[0..MAX_IDX_ZONE] OF REAL;
	cntTask : ARRAY[0..MAX_IDX_ZONE] OF UDINT;
	cntSamples : ARRAY[0..MAX_IDX_ZONE] OF UINT;
	HeatTest : Heat_Test_typ := (0);
	HeatSequence : ARRAY[0..MAX_IDX_TEMPGROUP] OF UINT := [MAX_IDX_TEMPGROUP+1(0)];
	HeatAlarm : Heat_Alarm_typ := (0);
	grp_TunePos : ARRAY[0..MAX_IDX_TEMPGROUP] OF BOOL;
	grp_TuneNeg : ARRAY[0..MAX_IDX_TEMPGROUP] OF BOOL;
	grp_PrePos : ARRAY[0..MAX_IDX_TEMPGROUP] OF BOOL;
	grp_PreNeg : ARRAY[0..MAX_IDX_TEMPGROUP] OF BOOL;
	grp_OnOffPos : ARRAY[0..MAX_IDX_TEMPGROUP] OF BOOL;
	grp_OnOffNeg : ARRAY[0..MAX_IDX_TEMPGROUP] OF BOOL;
	grpAct : UINT := 0;
	grpMaxIndex : UINT;
	grp : UINT := 0;
END_VAR
(*Heat  show Time*)
VAR
	uDisHeaterTime : UDINT;
	rHeaterTime : REAL;
END_VAR
(*Lowering Option*)
VAR
	bLowering : BOOL;
	TempUpLimit_HMI : ARRAY[0..MAX_IDX_ZONE] OF REAL;
	TempDwnLimit_HMI : ARRAY[0..MAX_IDX_ZONE] OF REAL;
	TempUpLimit_Same_HMI : REAL;
	TempDwnLimit_Same_HMI : REAL;
	TempInitOK : ARRAY[0..MAX_IDX_ZONE] OF REAL;
	bLowering_Hmi : BOOL;
	bLowering_Hmi_Pos : BOOL;
	TempInitOK_Old : ARRAY[0..MAX_IDX_ZONE] OF REAL;
	TempProtection : ARRAY[0..MAX_IDX_ZONE] OF REAL;
	TempProtectionFlag : BOOL;
	IsHeatPos : BOOL;
	TempProtectionMode : BOOL;
	TempProtectionFix_HMI : USINT;
	TempNotLow : ARRAY[0..MAX_IDX_ZONE] OF REAL;
	TempNotLowFlag : BOOL;
END_VAR
```

- edge.h (reference to Logical/GlobalIncludes/edge.h)

### Program Logical/Heating/h_pwm (ANSIC, version 1.00.0) - heating and cooling PWM

#### h_pwm.c - Implementation code
```c
/********************************************************************
 * COPYRIGHT --
 ********************************************************************
 * Program: h_pwm
 * File: h_pwm.c
 * Author: lijianjun
 * Created: March 04, 2013
 ********************************************************************
 * Implementation of program h_pwm --- heating and cooling PWM mode
 ********************************************************************/

#include <bur/plctypes.h>

#ifdef _DEFAULT_INCLUDES
	#include <AsDefault.h>
#endif

void _INIT h_pwmINIT(void)
{
	/* TODO: Add code here */
	gT_Par.GrpSwh.OnOff[0] = 0;
	for(ZoneIndex=0; ZoneIndex<MAX_IDX_CONTRL_ZONES; ZoneIndex++)
	{
		gT_Par.Ctl.OnOff[ZoneIndex] = 0;

		/* Heating time minum and Period  */
		gT_Par.Fix.tMinHeat[ZoneIndex]    = 0.05;
		gT_Par.Fix.tPeriodHeat[ZoneIndex] = 3.0;

        /* Cooling time minum and Period  */
		gT_Par.Fix.tMinCool[ZoneIndex]    = 0.2;
		gT_Par.Fix.tPeriodCool[ZoneIndex] = 3.0;

		LCRPWM_HeatArray[ZoneIndex].max_value = 100.0;
		LCRPWM_HeatArray[ZoneIndex].min_value = 0.0;

		LCRPWM_CoolArray[ZoneIndex].max_value = 100.0;
		LCRPWM_CoolArray[ZoneIndex].min_value = 0.0;
	}/* for(ZoneIndex=0; ZoneIndex<MAX_IDX_CONTRL_ZONES; ZoneIndex++) */
}

void _CYCLIC h_pwmCYCLIC(void)
{
	/* TODO: Add code here */

		/* quick setting parameters  */
		if(1 == gT_Par.Ctl.IsQuickSetValue && 0 == IsQuickSetValueOld)
		{
			gT_Par.Ctl.IsQuickSetValue = 0;
			for(ZoneIndex=0; ZoneIndex<MAX_IDX_ZONE; ZoneIndex++)
			{
				if(gT_Par.Par.ST_PID_Same > 0&& gT_Par.Par.ST_PID_Same <=gT_Par.Fix.AT_MAX)
				{
					gT_Par.Par.ST_PID[ZoneIndex] = gT_Par.Par.ST_PID_Same;
				}

				if(gT_Par.Par.AlaUpTol_Same > 0&& gT_Par.Par.AlaUpTol_Same <=gUserFix_new.TempUpRange)
				{
					gT_Par.Par.AlaUpTol[ZoneIndex] = gT_Par.Par.AlaUpTol_Same;
				}

				if(gT_Par.Par.AlaDwnTol_Same > 0&& gT_Par.Par.AlaDwnTol_Same <=gUserFix_new.TempDwnRange)
				{
					gT_Par.Par.AlaDwnTol[ZoneIndex] = gT_Par.Par.AlaDwnTol_Same;
				}
			}
		}/* if(1 == gT_Par.Ctl.IsQuickSetValue && 0 == IsQuickSetValueOld) */

		IsQuickSetValueOld = gT_Par.Ctl.IsQuickSetValue;

		bHeating = 0;
		for(ZoneIndex=0; ZoneIndex<MAX_IDX_CONTRL_ZONES; ZoneIndex++)
		{
			if(1 == gT_Par.Ctl.PreOnOff[ZoneIndex] || gT_Par.Ctl.OnOff[ZoneIndex])bHeating = 1;

			/* default heating pwm parameter */
			if(gT_Par.Fix.tMinHeat[ZoneIndex] < 0.05  )gT_Par.Fix.tMinHeat[ZoneIndex] = 0.05;
			if(1 == gT_Par.Fix.bContactor[ZoneIndex] && gT_Par.Fix.tMinHeat[ZoneIndex] < 0.3)gT_Par.Fix.tMinHeat[ZoneIndex] = 0.3;

			LCRPWM_HeatArray[ZoneIndex].enable = gT_Par.Fix.Enable[ZoneIndex];
			LCRPWM_HeatArray[ZoneIndex].t_min_pulse = gT_Par.Fix.tMinHeat[ZoneIndex];
			LCRPWM_HeatArray[ZoneIndex].t_period = gT_Par.Fix.tPeriodHeat[ZoneIndex];
			LCRPWM_HeatArray[ZoneIndex].x = gH_IO.y_heat[ZoneIndex];
			LCRPWM(&LCRPWM_HeatArray[ZoneIndex]);

			/* default cooling pwm parameter */
			if(gT_Par.Fix.tMinCool[ZoneIndex] < 0.3)gT_Par.Fix.tMinCool[ZoneIndex] = 0.3;
			gT_Par.Fix.tPeriodCool[ZoneIndex] = gT_Par.Fix.tPeriodHeat[ZoneIndex];

			LCRPWM_CoolArray[ZoneIndex].enable = gT_Par.Fix.Cooling[ZoneIndex];
			LCRPWM_CoolArray[ZoneIndex].t_min_pulse = gT_Par.Fix.tMinCool[ZoneIndex];
			LCRPWM_CoolArray[ZoneIndex].t_period = gT_Par.Fix.tPeriodCool[ZoneIndex];
			LCRPWM_CoolArray[ZoneIndex].x = gH_IO.y_cool[ZoneIndex];
			LCRPWM(&LCRPWM_CoolArray[ZoneIndex]);

			/* digital output  */
			gH_IO.do_H[ZoneIndex] = LCRPWM_HeatArray[ZoneIndex].pulse;
			gH_IO.do_C[ZoneIndex] = LCRPWM_CoolArray[ZoneIndex].pulse;

			/* analog output  */
			gH_IO.ao_H[ZoneIndex] = (INT)(gH_IO.y_heat[ZoneIndex] * 32767/100.0);
			gH_IO.ao_C[ZoneIndex] = (INT)(gH_IO.y_cool[ZoneIndex] * 32767/100.0);

			/* zones color  */

			if(1 == gT_Par.Status.SensorBroken[ZoneIndex])
			{
				gH_IO.ZoneColor[ZoneIndex] = 0x332A;	/* 红字黄底  *//*Word Red , Back Color Yellow*/
			}
			else if(1 == gT_Par.Status.AlmHigh[ZoneIndex])
			{
				gH_IO.ZoneColor[ZoneIndex] = 0x0137;   /* 蓝字红底  */	//*Word Blue , Back Color Red*/
			}
			else if(1 == gT_Par.Status.AlmLow[ZoneIndex])
			{
				gH_IO.ZoneColor[ZoneIndex] = 0x0110;	/* 蓝字白底  */	//*Word Blue , Back Color White*/
			}
			else
			{
				gH_IO.ZoneColor[ZoneIndex] = 0x0122;   /* 藍字黃底  */	//*Word Blue , Back Color Yellow*/
			}

			if(1 == gT_Par.Ctl.PreOnOff[ZoneIndex] )  /* 保温过程   */
			{
				gH_IO.ZoneColor[ZoneIndex] = 0x012F;   /* 蓝字黄底  */  //*Word Blue , Back Color Yellow*/
			}
			/***************************************************************************/
			/********************温区状态图组中的图片控制*******************************/
			/***************************************************************************/
			TON_StatusBG[ZoneIndex].IN = 1;

			if ((1 == gH_IO.do_H[ZoneIndex]) && (gH_IO.HC_sta[ZoneIndex] > 4))
			{
				gH_IO.HC_sta[ZoneIndex] = 4;
			}
			else if ((1 == gH_IO.do_C[ZoneIndex]) && (gH_IO.HC_sta[ZoneIndex] < 5))
			{
				gH_IO.HC_sta[ZoneIndex] = 5;
			}

			if (TON_StatusBG[ZoneIndex].Q == 1) 		/* 每1秒钟, 刷新图片 */
			{
				TON_StatusBG[ZoneIndex].IN = 0;

				if (1 ==gT_Par.Status.SensorBroken[ZoneIndex])
				{
					gH_IO.HC_sta[ZoneIndex] = 7;
				}
				else if (1 == gH_IO.do_H[ZoneIndex])
				{
					gH_IO.HC_sta[ZoneIndex] = gH_IO.HC_sta[ZoneIndex] + 1;

					if (gH_IO.HC_sta[ZoneIndex] > 4)
					{
						gH_IO.HC_sta[ZoneIndex] = 1;
					}
				}
				else if (1 == gH_IO.do_C[ZoneIndex])
				{
					gH_IO.HC_sta[ZoneIndex] = gH_IO.HC_sta[ZoneIndex] + 1;

					if (gH_IO.HC_sta[ZoneIndex] > 6)
					{
						gH_IO.HC_sta[ZoneIndex] = 5;
					}
				}
				else
				{
					gH_IO.HC_sta[ZoneIndex] = 0;
				}
			}/* if (TON_StatusBG[ZoneIndex].Q == 1) */

			/*********************************************************************************/
			/**************TON_StatusBG定时器实现*********************************************/
			/*********************************************************************************/
			TON_StatusBG[ZoneIndex].PT = 1000;				/*设定时间为1秒*/
			TON(&TON_StatusBG[ZoneIndex]);
		}/* for(ZoneIndex=0; ZoneIndex<MAX_IDX_CONTRL_ZONES; ZoneIndex++) */

		/* -------- 超溫保護開關 -------- */
		if(1 == gT_Par.Status.bSwitchOff)
		{
			gMachineOut.TempProtection = 1;
		}
		else
		{
			gMachineOut.TempProtection = 0;
		}
	}/* end of cyclic  */

void _EXIT h_pwmEXIT(void)
{
	/* TODO: Add code here */
}
```

#### h_pwm.var - Local variables
```iecst
(********************************************************************
 * COPYRIGHT --
 ********************************************************************
 * Program: h_pwm
 * File: h_pwm.var
 * Author: lij
 * Created: March 04, 2013
 ********************************************************************
 * Local variables of program h_pwm
 ********************************************************************)
VAR
	IsQuickSetValueOld : BOOL;
	bHeating : BOOL;
	ZoneIndex : UINT := 0;
	TON_StatusBG : ARRAY[0..MAX_IDX_ZONE] OF TON;
	LCRPWM_HeatArray : ARRAY[0..MAX_IDX_ZONE] OF LCRPWM := [MAX_IDX_ZONE+1(0)];
	LCRPWM_CoolArray : ARRAY[0..MAX_IDX_ZONE] OF LCRPWM := [MAX_IDX_ZONE+1(0)];
END_VAR
```

### Program Logical/Heating/trend (ANSIC, version 1.00.0) - temperature trend

#### trend.typ - Local data types
```iecst
(********************************************************************
 * COPYRIGHT --  B&R
 ********************************************************************
 * Program: trend
 * File: trend.typ
 * Author: lij
 * Created: March 06, 2013
 ********************************************************************
 * Local data types of program trend
 ********************************************************************)

TYPE
	Trend_typ : 	STRUCT
		Time_ScrollUp : BOOL;
		Time_ScrollDn : BOOL;
		Value_ScrollUp : BOOL;
		Value_ScrollDn : BOOL;
		Time_ZoomInc : BOOL;
		Time_ZoomDec : BOOL;
		Value_ZoomInc : BOOL;
		Value_ZoomDec : BOOL;
		Reset : BOOL;
		OldReset : BOOL;
		TimeMode : UINT;
		Time_Zoom : REAL;
		Value_Zoom : REAL;
		Time_Scroll : REAL;
		Value_Scroll : REAL;
		Cursor1Time : REAL;
		Cursor2Time : REAL;
		Curve : ARRAY[0..TREND_CURVE_NUM]OF Curve_typ;
END_STRUCT;
END_TYPE
```

#### trend.var
```iecst
VAR
	trend_1	:Trend_typ;
END_VAR
```

#### trend.c
```c
/********************************************************************
 * COPYRIGHT --  B&R
 ********************************************************************
 * Program: panel
 * File: panel.c
 * Author: lijianjun
 * Created: March 06, 2013
 ********************************************************************
 * Implementation of program panel --- display control
 ********************************************************************/

#include <bur/plctypes.h>
#include <string.h>

#ifdef _DEFAULT_INCLUDES
	#include <AsDefault.h>
#endif

#include "keyap2100.h"
//#include "keyap880.h"
#include "pic_id.h"

/**************************************************************************************
                            Function Declarations
**************************************************************************************/

void Trend( Trend_typ * pTrend);

/**************************************************************************************
     	        		I N I T U P  O F   T H E   T A S K
**************************************************************************************/
_INIT void init ( void )
{
	memset(&trend_1,0,sizeof(trend_1));

 	trend_1.Time_Zoom    = 1.0;
	trend_1.Value_Zoom   = 1.0;
	trend_1.Time_Scroll  = 0.0;
	trend_1.Value_Scroll = 0.0;

	trend_1.Curve[0].Status    = 1;
	trend_1.Curve[0].Value_Min = 0;
	trend_1.Curve[0].Value_Max = 300;

	trend_1.Curve[1].Status    = 1;
	trend_1.Curve[1].Value_Min = 0;
	trend_1.Curve[1].Value_Max = 300;

	trend_1.Curve[2].Status    = 1;
	trend_1.Curve[2].Value_Min = 0;
	trend_1.Curve[2].Value_Max = 300;

	trend_1.Curve[3].Status    = 1;
	trend_1.Curve[3].Value_Min = 0;
	trend_1.Curve[3].Value_Max = 300;

} /* end of _INIT */

 /*************************************************************************************
        				C Y C L I C   P A R T   O F   T H E   T A S K
**************************************************************************************/
 _CYCLIC void cyclic ( void )
{
	trend_1.Curve[0].Status = 0;
	trend_1.Curve[1].Status = 0;
	trend_1.Curve[2].Status = 0;
	trend_1.Curve[3].Status = 0;
	trend_1.Curve[4].Status = 0;

	if(gPanelObj.GetPicture == PIC_TEMP_TRACE_1 ||
	   gPanelObj.GetPicture == PIC_TEMP_TRACE_2 ||
	   gPanelObj.GetPicture == PIC_TEMP_TRACE_3 ||
	   gPanelObj.GetPicture == PIC_TEMP_TRACE_4 ||
	   gPanelObj.GetPicture == PIC_TEMP_TRACE_5)
	{
		trend_1.Reset         = gPanelObj.KeyMatric[S$KEYMATRIX_F8];
		trend_1.Time_ScrollDn = gPanelObj.KeyMatric[S$KEYMATRIX_F9];
		trend_1.Time_ScrollUp = gPanelObj.KeyMatric[S$KEYMATRIX_F10];
		trend_1.Value_ScrollDn = gPanelObj.KeyMatric[S$KEYMATRIX_F11];
		trend_1.Value_ScrollUp = gPanelObj.KeyMatric[S$KEYMATRIX_F12];
		trend_1.Value_ZoomDec = gPanelObj.KeyMatric[S$KEYMATRIX_F13];
		trend_1.Value_ZoomInc = gPanelObj.KeyMatric[S$KEYMATRIX_F14];

	}

	Trend(&trend_1);

}/* end of _CYCLIC */

void Trend( Trend_typ * pTrend)
{
	if(0 == pTrend->Reset && 1 == pTrend->OldReset)
	{
		pTrend->Time_Zoom    = 1.0;
		pTrend->Value_Zoom   = 1.0;
		pTrend->Time_Scroll  = 0.0;
		pTrend->Value_Scroll = 0.0;
	}

	pTrend->OldReset = pTrend->Reset;

	if(1 == pTrend->Value_ScrollUp)
	{
		pTrend->Value_Scroll = pTrend->Value_Scroll + 0.01;
	}

	if(1 == pTrend->Value_ScrollDn)
	{
		pTrend->Value_Scroll = pTrend->Value_Scroll - 0.01;
	}

	if(pTrend->Value_Scroll < -1.0)pTrend->Value_Scroll = -1.0;
	if(pTrend->Value_Scroll > 1.0)pTrend->Value_Scroll  = 1.0;

	if(1 == pTrend->Time_ScrollUp)
	{
		pTrend->Time_Scroll = pTrend->Time_Scroll + 0.01;
	}

	if(1 == pTrend->Time_ScrollDn)
	{
		pTrend->Time_Scroll = pTrend->Time_Scroll - 0.01;
	}

//	if(pTrend->Time_Scroll < -10.0)pTrend->Time_Scroll = -10.0;
//	if(pTrend->Time_Scroll > 10.0)pTrend->Time_Scroll  = 10.0;

	if(1 == pTrend->Value_ZoomInc)
	{
		pTrend->Value_Zoom = pTrend->Value_Zoom * 1.1;
	}

	if(1 == pTrend->Value_ZoomDec)
	{
		pTrend->Value_Zoom = pTrend->Value_Zoom * 0.9;
	}

	if(pTrend->Value_Zoom < 0.1 )pTrend->Value_Zoom = 0.1;
	if(pTrend->Value_Zoom > 10.0)pTrend->Value_Zoom = 10.0;

	if(1 == pTrend->Time_ZoomInc)
	{
		pTrend->Time_Zoom = pTrend->Time_Zoom * 1.1;
	}

	if(1 == pTrend->Time_ZoomDec)
	{
		pTrend->Time_Zoom = pTrend->Time_Zoom * 0.9;
	}

	if(pTrend->Time_Zoom < 0.1 )pTrend->Time_Zoom = 0.1;
	if(pTrend->Time_Zoom > 10.0)pTrend->Time_Zoom = 10.0;

}/*  void Trend( Trend_typ * pTrend) */
```

### Program Logical/Heating/h_plan (ANSIC, version 1.00.0) - heating time plan

#### h_plan.c - Implementation code
```c
/********************************************************************
 * COPYRIGHT --
 ********************************************************************
 * Program: h_plan
 * File: h_plan.c
 * Author: lijianjun
 * Created: March 06, 2013
 ********************************************************************
 * Implementation of program h_plan --- heating  plan
 ********************************************************************/

#include <bur/plctypes.h>

#ifdef _DEFAULT_INCLUDES
	#include <AsDefault.h>
#endif

void _INIT h_planINIT(void)
{
	/* TODO: Add code here */

}

void _CYCLIC h_planCYCLIC(void)
{
	/* TODO: Add code here */

	RTC_gettime(&rtGetTime);

	/*   week index     */
	if(rtGetTime.reserve > 7 || rtGetTime.reserve < 1)rtGetTime.reserve = 1;

	indexWeek = rtGetTime.reserve - 1;

	/*  預熱開   */
	if(1 == gHeatingPlan.Enable[indexWeek] && 1==gMachineIn.PreHeatDI)//ipis0220
	{
		if((rtGetTime.hour   == gHeatingPlan.HeatingOn[indexWeek].Hour  )&&
		   (rtGetTime.minute == gHeatingPlan.HeatingOn[indexWeek].Minute)&&
			(rtGetTime.second >0 && rtGetTime.second<3)
		  )
		{
			gT_Par.Ctl.IsPreHeatingPlan = 1;
		}
		else
		{
			gT_Par.Ctl.IsPreHeatingPlan = 0;
		}
	}/* if(1 == gHeatingPlan.Enable[indexWeek]) */
	else
	{
		gT_Par.Ctl.IsPreHeatingPlan = 0;
	}

	/*  加熱開   */
	if(1 == gHeatingPlan.Enable[7 + indexWeek])
	{
		if((rtGetTime.hour   == gHeatingPlan.HeatingOff[indexWeek].Hour  )&&
		   (rtGetTime.minute == gHeatingPlan.HeatingOff[indexWeek].Minute)&&
			(rtGetTime.second >0 && rtGetTime.second<3)
		  )
		{
			gT_Par.Ctl.IsHeatingOnPlan = 1;
		}
		else
		{
			gT_Par.Ctl.IsHeatingOnPlan = 0;
		}
	}/* if(1 == gHeatingPlan.Enable[7 + indexWeek]) */
	else
	{
		gT_Par.Ctl.IsHeatingOnPlan = 0;
	}

}
```

#### h_plan.var - Local variables
```iecst
(********************************************************************
 * COPYRIGHT --
 ********************************************************************
 * Program: h_plan
 * File: h_plan.var
 * Author: lij
 * Created: March 06, 2013
 ********************************************************************
 * Local variables of program h_plan
 ********************************************************************)
VAR
	indexWeek : USINT := 0;
	rtGetTime : RTCtime_typ := (0);
END_VAR
```

### Package Logical/spc - machine spc control

### spc.typ - Global data types
```iecst
(********************************************************************
 * COPYRIGHT --
 ********************************************************************
 * Package: spc
 * File: spc.typ
 * Author: lij
 * Created: July 15, 2015
 ********************************************************************
 * Data types of package spc
 ********************************************************************)

TYPE
	SPC_Ctrl_typ : 	STRUCT
		MoldL : SPC_Mold_Ctrl_typ;
		MoldR : SPC_Mold_Ctrl_typ;
	END_STRUCT;
	SPC_Par_typ : 	STRUCT
		UpperLimit : SPC_Unit_typ;
		LowerLimit : SPC_Unit_typ;
		CtrlEnable : SPC_Ctrl_typ;
	END_STRUCT;
	SPC_Screen_typ : 	STRUCT
		Data : ARRAY[0..23]OF SPC_Unit_typ;
		Max : SPC_Unit_typ;
		Avg : SPC_Unit_typ;
		Min : SPC_Unit_typ;
		Upper : SPC_Unit_typ;
		Lower : SPC_Unit_typ;
	END_STRUCT;
END_TYPE
```

### spc.var - Global variables
```iecst
(********************************************************************
 * COPYRIGHT --
 ********************************************************************
 * Package: spc
 * File: spc.var
 * Author: lij
 * Created: July 15, 2015
 ********************************************************************
 * Variables of package spc
 ********************************************************************)
VAR
	gSPC_Par : SPC_Par_typ;
END_VAR
```

### Program Logical/spc/spc_ctrl (ANSIC) - SPC data handling

#### spc_ctrl.c - Implementation code
```c
/********************************************************************
 * COPYRIGHT --
 ********************************************************************
 * Program: spc_ctrl
 * File: spc_ctrl.c
 * Author: lij
 * Created: July 16, 2015
 ********************************************************************
 * Implementation of program spc_ctrl
 ********************************************************************/

#include <bur/plctypes.h>
#include <string.h>

#ifdef _DEFAULT_INCLUDES
	#include <AsDefault.h>
#endif

#include "edge.h"
#include "keyap2100.h"
//#include "keyap880.h"
#include "pic_id.h"

#define S$MAX_SPC_NO 					 600	   /* Define Maximum Length of Quality Array is 600 */
#define S$SCREEN_SPC_NO 	    	    22		/* display Length of Quality Array is 22 */
/**************************************************************************************
** 							         function declare  				  			             **
**************************************************************************************/
void  SPC_Alarm();
void  SPC_Handle(UINT number);

/**************************************************************************************
**     	        		      I N I T U P  O F   T H E   T A S K 		 				       **
**************************************************************************************/

void _INIT spc_ctrlINIT(void)
{
	/* TODO: Add code here */
   strcpy(DataObjOperate.ModName,"spcdata");

   DataObjOperate.InitStep = 100;
   DataObjOperate.Step = 100;

}
/*************************************************************************************
**        				 C Y C L I C   P A R T   O F   T H E   T A S K  				   **
*************************************************************************************/
void _CYCLIC spc_ctrlCYCLIC(void)
{
	/* TODO: Add code here */
   int idx,i;
   /* --------------------	Step machine -- INIT -------------------- */
   switch(DataObjOperate.InitStep)
   {
      case 0:
         break;

      case 100:
         DatObj_Info.enable	= 1;
         DatObj_Info.pName	= (UDINT)DataObjOperate.ModName;

         /* Call  FUB  */
         DatObjInfo(&DatObj_Info);

         if (DatObj_Info.status == doERR_MODULNOTFOUND)	/* Data module not found -> create a new one */
         {
            DatObj_Info.enable = 0;
            DataObjOperate.InitStep  = 200;
         }
         else
         {
            DataObjOperate.Ident = DatObj_Info.ident;
            DataObjOperate.InitStep = 600;
         }
         break;

      case 200:
         /* Initialize create structure */
         DatObj_Create.enable = 1;
         DatObj_Create.grp	 	= 0;
         DatObj_Create.pName 	= (UDINT)DataObjOperate.ModName;
         DatObj_Create.len 	= sizeof(SPC_Unit_typ)* (S$MAX_SPC_NO + S$SCREEN_SPC_NO)+ sizeof(idxSPC);
         DatObj_Create.MemType  = doUSRROM;
         DatObj_Create.Option   = 0;
         DatObj_Create.pCpyData = 0;

         /* Call FUB */
         DatObjCreate(&DatObj_Create);

         /* Get FUB output information */
         if( 0 == DatObj_Create.status)
         {
            DatObj_Create.enable = 0;
            DataObjOperate.Ident = DatObj_Create.ident;
            DataObjOperate.InitStep = 300;
         }
         break;

      case 300:
         status_tmpalloc = TMP_alloc(sizeof(SPC_Unit_typ)* (S$MAX_SPC_NO + S$SCREEN_SPC_NO) + sizeof(idxSPC), (void*)&pData);
         if(0 == status_tmpalloc)
         {
            memset((void*)pData,0,sizeof(SPC_Unit_typ)* (S$MAX_SPC_NO + S$SCREEN_SPC_NO) + sizeof(idxSPC));
            DataObjOperate.InitStep = 400;
         }
         else
         {
            DataObjOperate.InitStep = 9999;
         }
         break;

      case 400:
         DatObj_Write.enable  = 1;
         DatObj_Write.ident 	= DataObjOperate.Ident;
         DatObj_Write.Offset  = 0;
         DatObj_Write.pSource = (UDINT)pData;
         DatObj_Write.len 	= sizeof(SPC_Unit_typ)* (S$MAX_SPC_NO + S$SCREEN_SPC_NO) + sizeof(idxSPC);

         /* Call FUB */
         DatObjWrite(&DatObj_Write);

         if(0 == DatObj_Write.status)
         {
            DatObj_Write.enable = 0;
            DataObjOperate.InitStep = 500;
         }
         break;

      case 500:
         status_tmpfree = TMP_free(sizeof(SPC_Unit_typ)* (S$MAX_SPC_NO + S$SCREEN_SPC_NO) + sizeof(idxSPC), (void*)pData);
         if(0 == status_tmpfree)
         {
            DataObjOperate.InitStep = 600;
         }
         else
         {
            DataObjOperate.InitStep = 9999;
         }
         break;

      case 600:
         DatObj_Read.enable = 1;
         DatObj_Read.ident  = DataObjOperate.Ident;
         DatObj_Read.Offset = 0;
         DatObj_Read.pDestination = (UDINT)&idxSPC;
         DatObj_Read.len = sizeof(idxSPC);

         /* Call FUB */
         DatObjRead(&DatObj_Read);
         if(0 == DatObj_Read.status)
			{
				oldCycleNo = gCycleTimes;
				gSPC_Current.CycleNo = gCycleTimes;
				DatObj_Read.enable = 0;

				if(idxSPC >= 0 && idxSPC < 2 * S$MAX_SPC_NO)
				{
					DataObjOperate.InitStep = 3000;
				}
				else
				{
					DataObjOperate.InitStep = 300;  /* init value  */
				}
			}
         else
         {
            DataObjOperate.InitStep = 9999;
         }
         break;

      case 3000:
         break;

      case 9999:
         DataObjOperate.InitStep = 0;
         break;
   }/* switch(DataObjOperate.InitStep) */

   if(DataObjOperate.Ident == 0 || DataObjOperate.InitStep != 3000)
   {
      return;
   }/* if(DataObjOperate.Ident == 0 || DataObjOperate.InitStep != 3000) */

   if(PIC_SPC_CTRL == gPanelObj.GetPicture)
   {
      for(i=0;i<sizeof(SPC_Mold_Ctrl_typ);i++)
      {
         if(16384 == FocusCtrlL[i])
         {
            if(1 == EDGEPOS(gPanelObj.KeyMatric[S$KEYMATRIX_TAB],KeyMatric[S$KEYMATRIX_TAB]))
            {
               ((USINT *)(&gSPC_Par.CtrlEnable.MoldL.tCycle))[i] = !((USINT *)(&gSPC_Par.CtrlEnable.MoldL.tCycle))[i];
               gRecipeOperate.OnceSave = 1;
            }
         }

         if(16384 == FocusCtrlR[i])
         {
            if(1 == EDGEPOS(gPanelObj.KeyMatric[S$KEYMATRIX_TAB],KeyMatric[S$KEYMATRIX_TAB]))
            {
               ((USINT *)(&gSPC_Par.CtrlEnable.MoldR.tCycle))[i] = !((USINT *)(&gSPC_Par.CtrlEnable.MoldR.tCycle))[i];
               gRecipeOperate.OnceSave = 1;
            }
         }
      }
   }
   KeyMatric[S$KEYMATRIX_TAB] = gPanelObj.KeyMatric[S$KEYMATRIX_TAB];

   /* SPC oil temperature  */
   gSPC_Current.OilTemp = gMachineInfo.OilTemp;

   /* cycle change  */
   gSPC_Current.CycleNo = gCycleTimes;

   if(oldCycleNo != gSPC_Current.CycleNo)
   {
      bCycleChange = 1;
   }

   oldCycleNo = gSPC_Current.CycleNo;

   /*  call function  */
   SPC_Alarm();

   if(gPanelObj.GetPicture != PIC_SPC_1 && gPanelObj.GetPicture != PIC_SPC_2 &&
      gPanelObj.GetPicture != PIC_SPC_CTRL)
   {
      bCmdRefresh = 1;
   }

   /* ------------- step machine ctrl ------------- */
   switch(DataObjOperate.Step )
   {
      case 100:
         if(1 == bCycleChange)
         {
            bCycleChange = 0;
            DataObjOperate.Step = 1000;
         }/* if(1 == bCycleChange) */
         else
         {
            if(gPanelObj.GetPicture == PIC_SPC_1 || gPanelObj.GetPicture == PIC_SPC_2 ||
               gPanelObj.GetPicture == PIC_SPC_CTRL)
            {
               if(1 == bCmdRefresh)
               {
                  bCmdRefresh = 0;
                  idxScreen  = idxSPC;
                  DataObjOperate.Step = 2000;
               }
            }

            if(gPanelObj.GetPicture == PIC_SPC_1 || gPanelObj.GetPicture == PIC_SPC_2)
            {
               if(1 == EDGEPOS(gPanelObj.KeyMatric[S$KEYMATRIX_F7],KeyMatric[S$KEYMATRIX_F7]))
					{
						if((idxScreen % S$MAX_SPC_NO) >= S$SCREEN_SPC_NO)idxScreen = idxScreen - S$SCREEN_SPC_NO;
						if(idxScreen > 0 && idxScreen < 2 * S$MAX_SPC_NO)
						{
							DataObjOperate.Step = 2000;
						}
					}

               if(1 == EDGEPOS(gPanelObj.KeyMatric[S$KEYMATRIX_F8],KeyMatric[S$KEYMATRIX_F8]))
					{
						if((idxScreen % S$MAX_SPC_NO) < S$MAX_SPC_NO - S$SCREEN_SPC_NO)idxScreen = idxScreen + S$SCREEN_SPC_NO;
						if(idxScreen > 0 && idxScreen < 2 * S$MAX_SPC_NO)
						{
							DataObjOperate.Step = 2000;
						}
					}
            }/* if(gPanelObj.GetPicture == PIC_SPC_1 || gPanelObj.GetPicture == PIC_SPC_2) */
         }/* if(1 == bCycleChange) */
         break;

      case 1000:
         DatObj_Write.enable  = 1;
         DatObj_Write.ident	= DataObjOperate.Ident;

         DatObj_Write.Offset  = sizeof(gSPC_Current) * (idxSPC % S$MAX_SPC_NO) + sizeof(idxSPC);
         DatObj_Write.pSource = (UDINT)(&gSPC_Current);
         DatObj_Write.len     = sizeof(gSPC_Current);

         DatObjWrite(&DatObj_Write);
         if(0 == DatObj_Write.status)
         {
            DatObj_Write.enable = 0;

			if(1 == gSPC_Current.MoldR.bCleanCycle)
			{
				memset(&gSPC_Current.MoldR,0,sizeof(gSPC_Current.MoldR));
			}
			else if(1 == gSPC_Current.MoldL.bCleanCycle)
			{
				memset(&gSPC_Current.MoldL,0,sizeof(gSPC_Current.MoldL));
			}

            DataObjOperate.Step = 1100;
         }
         break;

		//SPC CleanCycle
//		case 1050:
//			if(1 == gSPC_Current.MoldR.bCleanCycle)
//			{
//				memset(&gSPC_Current.MoldR,0,sizeof(gSPC_Current.MoldR));
//			}
//			else if(1 == gSPC_Current.MoldL.bCleanCycle)
//			{
//				memset(&gSPC_Current.MoldL,0,sizeof(gSPC_Current.MoldL));
//			}
//			DataObjOperate.Step = 1100;
//			break;

      case 1100:
         if((idxSPC % S$MAX_SPC_NO) < S$SCREEN_SPC_NO)
         {
            DataObjOperate.Step = 1200;
         }
         else
         {
            DataObjOperate.Step = 1300;
         }
         break;

      case 1200:
         DatObj_Write.enable  = 1;
         DatObj_Write.ident	 = DataObjOperate.Ident;

         DatObj_Write.Offset  = sizeof(gSPC_Current) * ((idxSPC % S$MAX_SPC_NO) + S$MAX_SPC_NO)+ sizeof(idxSPC);
         DatObj_Write.pSource = (UDINT)(&gSPC_Current);
         DatObj_Write.len     = sizeof(gSPC_Current);

         DatObjWrite(&DatObj_Write);
         if(0 == DatObj_Write.status)
         {
            DatObj_Write.enable = 0;

			if(1 == gSPC_Current.MoldR.bCleanCycle)
			{
				memset(&gSPC_Current.MoldR,0,sizeof(gSPC_Current.MoldR));
			}
			else if(1 == gSPC_Current.MoldL.bCleanCycle)
			{
				memset(&gSPC_Current.MoldL,0,sizeof(gSPC_Current.MoldL));
			}

            DataObjOperate.Step = 1300;
         }
         break;

		//SPC clean
//	  case 1250:
//			if(1 == gSPC_Current.MoldR.bCleanCycle)
//			{
//				memset(&gSPC_Current.MoldR,0,sizeof(gSPC_Current.MoldR));
//			}
//			else if(1 == gSPC_Current.MoldL.bCleanCycle)
//			{
//				memset(&gSPC_Current.MoldL,0,sizeof(gSPC_Current.MoldL));
//			}
//			DataObjOperate.Step = 1300;
//		 break;

      case 1300:
         idxSPC = idxSPC + 1;
         if(idxSPC >= 2 * S$MAX_SPC_NO)idxSPC = S$MAX_SPC_NO;
         DataObjOperate.Step = 1400;
         break;

      case 1400:
         DatObj_Write.enable  = 1;
         DatObj_Write.ident	 = DataObjOperate.Ident;

         DatObj_Write.Offset  = 0;
         DatObj_Write.pSource = (UDINT)(&idxSPC);
         DatObj_Write.len     = sizeof(idxSPC);

         DatObjWrite(&DatObj_Write);
         if(0 == DatObj_Write.status)
         {
            DatObj_Write.enable = 0;
            DataObjOperate.Step = 1500;
         }
         break;

      case 1500:
         idxScreen  = idxSPC;
         DataObjOperate.Step = 2000;
         break;

      case 2000:
         memset(&DataList[0],0,sizeof(DataList));
         if(0 == idxScreen)
         {
            DataObjOperate.Step = 5000;
         }
         else if(idxScreen <= S$SCREEN_SPC_NO)
         {
            DataObjOperate.Step = 2100;
         }
         else if(idxScreen > S$SCREEN_SPC_NO)
         {
            DataObjOperate.Step = 2600;
         }
         break;

      case 2100:
         DatObj_Read.enable = 1;
         DatObj_Read.ident  = DataObjOperate.Ident;

         DatObj_Read.Offset = sizeof(idxSPC);
         DatObj_Read.pDestination = (UDINT)&DataList;
         DatObj_Read.len = sizeof(gSPC_Current) * idxScreen;

         /* Call FUB */
         DatObjRead(&DatObj_Read);
         if(0 == DatObj_Read.status)
         {
            DatObj_Read.enable = 0;
            DataObjOperate.Step = 2200;
         }
         break;

      case 2200:
         for(idx=0;idx<idxScreen;idx++)
         {
            SPC_Dis.Data[idxScreen -1 - idx]= DataList[idx];
         }
         DataObjOperate.Step = 2300;
         break;

      case 2300:
         SPC_Dis.Max = SPC_Dis.Data[0];
         SPC_Dis.Min = SPC_Dis.Data[0];
         memset(&SPC_Dis.Avg,0,sizeof(SPC_Dis.Avg));
         SPC_Handle(idxScreen);

         DataObjOperate.Step = 2400;
         break;

      case 2400:
         DataObjOperate.Step = 100;
         break;

      case 2600:
         DatObj_Read.enable = 1;
         DatObj_Read.ident  = DataObjOperate.Ident;

         if(idxScreen < (S$MAX_SPC_NO + S$SCREEN_SPC_NO))
         {
            DatObj_Read.Offset = (idxScreen - S$SCREEN_SPC_NO) * sizeof(gSPC_Current) + sizeof(idxSPC);
         }
         else
         {
            DatObj_Read.Offset = ((idxScreen % S$MAX_SPC_NO) - S$SCREEN_SPC_NO) * sizeof(gSPC_Current)+ sizeof(idxSPC);
         }
         DatObj_Read.pDestination = (UDINT)&DataList;
         DatObj_Read.len = sizeof(gSPC_Current) * S$SCREEN_SPC_NO;

         /* Call FUB */
         DatObjRead(&DatObj_Read);
         if(0 == DatObj_Read.status)
         {
            DatObj_Read.enable = 0;
            DataObjOperate.Step = 2700;
         }
         break;

      case 2700:
         for(idx=0;idx<S$SCREEN_SPC_NO;idx++)
         {
            SPC_Dis.Data[S$SCREEN_SPC_NO - 1 - idx]= DataList[idx];
         }
         DataObjOperate.Step = 2800;
         break;

      case 2800:
         SPC_Dis.Max = SPC_Dis.Data[0];
         SPC_Dis.Min = SPC_Dis.Data[0];
         memset(&SPC_Dis.Avg,0,sizeof(SPC_Dis.Avg));

         SPC_Handle(S$SCREEN_SPC_NO);

         DataObjOperate.Step = 2900;
         break;

      case 2900:
         DataObjOperate.Step = 100;
         break;

      case 5000:
         DataObjOperate.Step = 100;
         break;
      default:
         break;
   }/* switch(DataObjOperate.Step) */

   oldPicture = gPanelObj.GetPicture;
}

void _EXIT spc_ctrlEXIT(void)
{
	/* TODO: Add code here */
}

void  SPC_Alarm()
{
   int idx;

   for(idx=0;idx<sizeof(SPC_Mold_Ctrl_typ);idx++)
   {
      if(1 == ((USINT *)(&gSPC_Par.CtrlEnable.MoldL.tCycle))[idx]) /*   */
      {
         if(((REAL *)(&gSPC_Current.MoldL.tCycle))[idx] > ((REAL *)(&gSPC_Par.UpperLimit.MoldL.tCycle))[idx])
         {
            ((USINT *)(&gAlarm.UpperLSPC.tCycle))[idx] = 1;
         }

         if(((REAL *)(&gSPC_Current.MoldL.tCycle))[idx] > ((REAL *)(&gSPC_Par.LowerLimit.MoldL.tCycle))[idx])
         {
            ((USINT *)(&gAlarm.LowerLSPC.tCycle))[idx] = 1;
         }
      }
      else
      {
         ((USINT *)(&gAlarm.UpperLSPC.tCycle))[idx] = 0;
         ((USINT *)(&gAlarm.LowerLSPC.tCycle))[idx] = 0;
      }

      if(1 == ((USINT *)(&gSPC_Par.CtrlEnable.MoldR.tCycle))[idx])
      {
         if(((REAL *)(&gSPC_Current.MoldR.tCycle))[idx] > ((REAL *)(&gSPC_Par.UpperLimit.MoldR.tCycle))[idx])
         {
            ((USINT *)(&gAlarm.UpperRSPC.tCycle))[idx] = 1;
         }

         if(((REAL *)(&gSPC_Current.MoldR.tCycle))[idx] > ((REAL *)(&gSPC_Par.LowerLimit.MoldR.tCycle))[idx])
         {
            ((USINT *)(&gAlarm.LowerRSPC.tCycle))[idx] = 1;
         }
      }
      else
      {
         ((USINT *)(&gAlarm.UpperRSPC.tCycle))[idx] = 0;
         ((USINT *)(&gAlarm.LowerRSPC.tCycle))[idx] = 0;
      }
   }/* for(idx=0;idx<sizeof(gSPC_Par.CtrlEnable.MoldL);idx++) */
}/* void  SPC_Alarm() */

void  SPC_Handle(UINT number)
{
   int idx,idxValue;

   for(idx=0;idx<number;idx++)
   {
      if(SPC_Dis.Max.OilTemp < SPC_Dis.Data[idx].OilTemp)SPC_Dis.Max.OilTemp = SPC_Dis.Data[idx].OilTemp;
      if(SPC_Dis.Min.OilTemp > SPC_Dis.Data[idx].OilTemp)SPC_Dis.Min.OilTemp = SPC_Dis.Data[idx].OilTemp;
      SPC_Dis.Avg.OilTemp = SPC_Dis.Avg.OilTemp + SPC_Dis.Data[idx].OilTemp/number;

      for(idxValue=0;idxValue<sizeof(SPC_Mold_Ctrl_typ);idxValue++)
      {
         /*  left mold value   */
         if(((REAL *)(&SPC_Dis.Max.MoldL.tCycle))[idxValue] < ((REAL *)(&SPC_Dis.Data[idx].MoldL.tCycle))[idxValue])
         {
            ((REAL *)(&SPC_Dis.Max.MoldL.tCycle))[idxValue] = ((REAL *)(&SPC_Dis.Data[idx].MoldL.tCycle))[idxValue];
         }

         if(((REAL *)(&SPC_Dis.Min.MoldL.tCycle))[idxValue] > ((REAL *)(&SPC_Dis.Data[idx].MoldL.tCycle))[idxValue])
         {
            ((REAL *)(&SPC_Dis.Min.MoldL.tCycle))[idxValue] = ((REAL *)(&SPC_Dis.Data[idx].MoldL.tCycle))[idxValue];
         }

         ((REAL *)(&SPC_Dis.Avg.MoldL.tCycle))[idxValue] = ((REAL *)(&SPC_Dis.Avg.MoldL.tCycle))[idxValue] +
                                                           ((REAL *)(&SPC_Dis.Data[idx].MoldL.tCycle))[idxValue]/number;

         /*  right mold value   */
         if(((REAL *)(&SPC_Dis.Max.MoldR.tCycle))[idxValue] < ((REAL *)(&SPC_Dis.Data[idx].MoldR.tCycle))[idxValue])
         {
            ((REAL *)(&SPC_Dis.Max.MoldR.tCycle))[idxValue] = ((REAL *)(&SPC_Dis.Data[idx].MoldR.tCycle))[idxValue];
         }

         if(((REAL *)(&SPC_Dis.Min.MoldR.tCycle))[idxValue] > ((REAL *)(&SPC_Dis.Data[idx].MoldR.tCycle))[idxValue])
         {
            ((REAL *)(&SPC_Dis.Min.MoldR.tCycle))[idxValue] = ((REAL *)(&SPC_Dis.Data[idx].MoldR.tCycle))[idxValue];
         }

         ((REAL *)(&SPC_Dis.Avg.MoldR.tCycle))[idxValue] = ((REAL *)(&SPC_Dis.Avg.MoldR.tCycle))[idxValue] +
                                                           ((REAL *)(&SPC_Dis.Data[idx].MoldR.tCycle))[idxValue]/number;
      }/* for(idxValue=0;idxValue<sizeof(SPC_Mold_Ctrl_typ);idxValue++) */
   }/* for(idx=0;idx<number;idx++) */
}/* void  SPC_Handle(UINT number) */
```

#### spc_ctrl.var - Local variables
```iecst
(********************************************************************
 * COPYRIGHT --
 ********************************************************************
 * Program: spc_ctrl
 * File: spc_ctrl.var
 * Author: lij
 * Created: July 16, 2015
 ********************************************************************
 * Local variables of program spc_ctrl
 ********************************************************************)
VAR
	KeyMatric : ARRAY[0..99] OF USINT;
	DataObjOperate : DatObj_Operate_typ;
	DatObj_Info : DatObjInfo;
	DatObj_Create : DatObjCreate;
	DatObj_Write : DatObjWrite;
	DatObj_Read : DatObjRead;
	idxSPC : UDINT;
	pData : UDINT;
	status_tmpalloc : UINT;
	status_tmpfree : UINT;
	oldCycleNo : UDINT;
	bCycleChange : BOOL;
	bCmdRefresh : BOOL;
	idxScreen : UDINT;
	SPC_Dis : SPC_Screen_typ;
	DataList : ARRAY[0..23] OF SPC_Unit_typ;
	FocusCtrlL : ARRAY[0..19] OF UINT;
	FocusCtrlR : ARRAY[0..19] OF UINT;
	oldPicture : UINT;
END_VAR
```

- pic_id.h (reference to Logical/GlobalIncludes/pic_id.h)

- keyap880.h (reference to Logical/GlobalIncludes/keyap880.h)

### Package Logical/ThirdDrive - 3nd dirve control using motorkey

### Program Logical/ThirdDrive/axisctrl (ANSIC, version 1.00.0) - 3nd servo motor control

#### axisctrl.c
```c
/********************************************************************
 * COPYRIGHT -- B&R China
 ********************************************************************
 * Program: axisctrl
 * File: axisctrl.c
 * Author: lijianjun
 * Created: March 06, 2013
 ********************************************************************
 * Implementation of program axisctrl --- Third servo drive axis control
 ********************************************************************/
#include <bur/plctypes.h>
#include <string.h>

#ifdef _DEFAULT_INCLUDES
	#include <AsDefault.h>
#endif

#define	STATE_WAIT				 0
#define	STATE_POWER_ON			10
#define	STATE_INIT_HOME		20

#define	STATE_READY				100

#define	STATE_HOME				110
#define	STATE_STOP				120
#define	STATE_MOVE_JOG_POS	130
#define	STATE_MOVE_JOG_NEG	140
#define	STATE_MOVE_ABSOLUTE	150
#define	STATE_MOVE_RELATIVE	160

#define	STATE_ERROR				210
#define	STATE_ERROR_RESET		220
/**************************************************************************************
**     	        		I N I T U P  O F   T H E   T A S K 		 				     **
**************************************************************************************/
_INIT void axisctrl_init(void)
{

	for(idxAxis=0;idxAxis<MAX_AXIS_NUM;idxAxis++)
	{
		gDS1119_Axis[idxAxis].init.taskTime = 0.002;    /* 2ms task time   */
		gDS1119_Axis[idxAxis].init.units = 1250;		/* 12.5mm * 100/rev  */
		gDS1119_Axis[idxAxis].init.microsteps = 10000;		/* 10000 pulse /rev   */
		gDS1119_Axis[idxAxis].init.reverseDirection = 1;

		gAxisCtrl[idxAxis].param.speed = 3000;
		gAxisCtrl[idxAxis].param.acceleration = 187500;
		gAxisCtrl[idxAxis].param.deceleration = 187500;

		gAxisCtrl[idxAxis].step = STATE_WAIT;
		gAxisCtrl[idxAxis].cmd.power = 1;
		gAxisCtrl[idxAxis].bHomeOk = 0;
	}
}/* end of _INIT */

/*************************************************************************************
**        				C Y C L I C   P A R T   O F   T H E   T A S K  				**
*************************************************************************************/
_CYCLIC void axisctrl_cyc(void)
{
	/*DS1119_1_OK = gDS1119_Axis[0].IOMapping.ModuleOk;
	DS1119_2_OK = gDS1119_Axis[1].IOMapping.ModuleOk;*/

	for(idxAxis=0;idxAxis<MAX_AXIS_NUM;idxAxis++)
	{
		/* default speed  */
		if(0 == gAxisCtrl[idxAxis].param.speed)gAxisCtrl[idxAxis].param.speed = 3000;

		gAxisCtrl[idxAxis].As = gDS1119_Axis[idxAxis].info.position/100.0;
		/* step machine control  */
		switch(gAxisCtrl[idxAxis].step)
		{
			case STATE_WAIT:
				gAxisCtrl[idxAxis].cmd.homing = 0;
				gAxisCtrl[idxAxis].cmd.stop   = 0;
				gAxisCtrl[idxAxis].cmd.jogPos   = 0;
				gAxisCtrl[idxAxis].cmd.jogNeg   = 0;
				gAxisCtrl[idxAxis].cmd.absolute = 0;
				gAxisCtrl[idxAxis].cmd.relative = 0;
				gAxisCtrl[idxAxis].cmd.acknowledge = 0;

				gDS1119_Axis[idxAxis].cmd.homing = 0;
				gDS1119_Axis[idxAxis].cmd.stop   = 0;
				gDS1119_Axis[idxAxis].cmd.absolute = 0;
				gDS1119_Axis[idxAxis].cmd.additive = 0;
				gDS1119_Axis[idxAxis].cmd.velocity= 0;
				gDS1119_Axis[idxAxis].cmd.acknowledge = 0;

				if(1 == gDS1119_Axis[idxAxis].info.initialized)
				{
					if(1 == gAxisCtrl[idxAxis].cmd.power)
					{
						gDS1119_Axis[idxAxis].cmd.power = 1;
						gAxisCtrl[idxAxis].step = STATE_POWER_ON;
					}

					gDS1119_Axis[idxAxis].cmd.homing = 0;
				}
				break;
			case STATE_POWER_ON:
				if(1 == gDS1119_Axis[idxAxis].info.powerOn)
				{
					gDS1119_Axis[idxAxis].cmd.homing = 1;
					gAxisCtrl[idxAxis].step = STATE_INIT_HOME;
				}

				if(gDS1119_Axis[idxAxis].info.status != 0)
				{
					gAxisCtrl[idxAxis].errorID = gDS1119_Axis[idxAxis].info.status;
					strcpy(gAxisCtrl[idxAxis].errorText,gDS1119_Axis[idxAxis].info.errorText);
					gAxisCtrl[idxAxis].step = STATE_ERROR;
				}
				break;

			case STATE_INIT_HOME:
				if(1 == gDS1119_Axis[idxAxis].info.homingOk)
				{
					if(1 == gAxisCtrl[idxAxis].bRefer)
					{
						gAxisCtrl[idxAxis].bHomeOk = 1;
					}

					gAxisCtrl[idxAxis].step = STATE_READY;
				}

				if(gDS1119_Axis[idxAxis].info.status != 0)
				{
					gAxisCtrl[idxAxis].errorID = gDS1119_Axis[idxAxis].info.status;
					strcpy(gAxisCtrl[idxAxis].errorText,gDS1119_Axis[idxAxis].info.errorText);
					gAxisCtrl[idxAxis].step = STATE_ERROR;
				}
				break;

			case STATE_READY:
				if(1 == gAxisCtrl[idxAxis].cmd.homing)
				{
					gAxisCtrl[idxAxis].cmd.homing  = 0;
					gDS1119_Axis[idxAxis].cmd.homing = 1;
					gAxisCtrl[idxAxis].step = STATE_HOME;
				}
				else if(1 == gAxisCtrl[idxAxis].cmd.stop)
				{
					gAxisCtrl[idxAxis].cmd.stop = 0;
					gDS1119_Axis[idxAxis].cmd.stop = 1;
					gDS1119_Axis[idxAxis].param.deceleration = gAxisCtrl[idxAxis].param.deceleration;

					gAxisCtrl[idxAxis].step = STATE_STOP;
				}
				else if(1 == gAxisCtrl[idxAxis].cmd.jogPos)
				{
					gDS1119_Axis[idxAxis].cmd.velocity = gAxisCtrl[idxAxis].cmd.jogPos;
					gDS1119_Axis[idxAxis].param.speed  = gAxisCtrl[idxAxis].param.speed;
					gDS1119_Axis[idxAxis].param.acceleration = gAxisCtrl[idxAxis].param.acceleration;
					gDS1119_Axis[idxAxis].param.deceleration = gAxisCtrl[idxAxis].param.deceleration;

					gAxisCtrl[idxAxis].step = STATE_MOVE_JOG_POS;
				}
				else if(1 == gAxisCtrl[idxAxis].cmd.jogNeg)
				{
					gDS1119_Axis[idxAxis].cmd.velocity = gAxisCtrl[idxAxis].cmd.jogNeg;
					gDS1119_Axis[idxAxis].param.speed  = -gAxisCtrl[idxAxis].param.speed;
					gDS1119_Axis[idxAxis].param.acceleration = gAxisCtrl[idxAxis].param.acceleration;
					gDS1119_Axis[idxAxis].param.deceleration = gAxisCtrl[idxAxis].param.deceleration;

					gAxisCtrl[idxAxis].step = STATE_MOVE_JOG_NEG;
				}
				else if(1 == gAxisCtrl[idxAxis].cmd.absolute)
				{
					gAxisCtrl[idxAxis].cmd.absolute  = 0;
					gDS1119_Axis[idxAxis].cmd.absolute = 1;
					gDS1119_Axis[idxAxis].param.position = gAxisCtrl[idxAxis].param.position;
					gDS1119_Axis[idxAxis].param.speed    = gAxisCtrl[idxAxis].param.speed;
					gDS1119_Axis[idxAxis].param.acceleration = gAxisCtrl[idxAxis].param.acceleration;
					gDS1119_Axis[idxAxis].param.deceleration = gAxisCtrl[idxAxis].param.deceleration;

					gAxisCtrl[idxAxis].step = STATE_MOVE_ABSOLUTE;
				}
				else if(1 == gAxisCtrl[idxAxis].cmd.relative)
				{
					gAxisCtrl[idxAxis].cmd.relative = 0;
					gDS1119_Axis[idxAxis].cmd.additive = 1;
					gDS1119_Axis[idxAxis].param.position = gAxisCtrl[idxAxis].param.position;
					gDS1119_Axis[idxAxis].param.speed    = gAxisCtrl[idxAxis].param.speed;
					gDS1119_Axis[idxAxis].param.acceleration = gAxisCtrl[idxAxis].param.acceleration;
					gDS1119_Axis[idxAxis].param.deceleration = gAxisCtrl[idxAxis].param.deceleration;

					gAxisCtrl[idxAxis].step = STATE_MOVE_RELATIVE;
				}
				break;

			case STATE_HOME:
				if(1 == gDS1119_Axis[idxAxis].info.homingOk)
				{
					if(1 == gAxisCtrl[idxAxis].bRefer)
					{
						gAxisCtrl[idxAxis].bHomeOk = 1;
					}

					gAxisCtrl[idxAxis].step = STATE_READY;
				}

				if(gDS1119_Axis[idxAxis].info.status != 0)
				{
					gAxisCtrl[idxAxis].errorID = gDS1119_Axis[idxAxis].info.status;
					strcpy(gAxisCtrl[idxAxis].errorText,gDS1119_Axis[idxAxis].info.errorText);
					gAxisCtrl[idxAxis].step = STATE_ERROR;
				}
				break;

			case STATE_STOP:
				gDS1119_Axis[idxAxis].param.deceleration = gAxisCtrl[idxAxis].param.deceleration;

				if(0 == gDS1119_Axis[idxAxis].info.moveActive)
				{
					gAxisCtrl[idxAxis].step = STATE_READY;
				}

				if(gDS1119_Axis[idxAxis].info.status != 0)
				{
					gAxisCtrl[idxAxis].errorID = gDS1119_Axis[idxAxis].info.status;
					strcpy(gAxisCtrl[idxAxis].errorText,gDS1119_Axis[idxAxis].info.errorText);
					gAxisCtrl[idxAxis].step = STATE_ERROR;
				}
				break;

			case STATE_MOVE_JOG_POS:
				gDS1119_Axis[idxAxis].cmd.velocity = gAxisCtrl[idxAxis].cmd.jogPos;

				gDS1119_Axis[idxAxis].param.speed  = gAxisCtrl[idxAxis].param.speed;
				gDS1119_Axis[idxAxis].param.acceleration = gAxisCtrl[idxAxis].param.acceleration;
				gDS1119_Axis[idxAxis].param.deceleration = gAxisCtrl[idxAxis].param.deceleration;

				if(1 == gAxisCtrl[idxAxis].cmd.stop)
				{
					gAxisCtrl[idxAxis].cmd.stop   = 0;
					gAxisCtrl[idxAxis].cmd.jogPos = 0;
					gDS1119_Axis[idxAxis].cmd.velocity = 0;
					gDS1119_Axis[idxAxis].cmd.stop     = 1;
					gAxisCtrl[idxAxis].step = STATE_STOP;
				}
				else if(0 == gDS1119_Axis[idxAxis].cmd.velocity)
				{
					if(0 == gDS1119_Axis[idxAxis].info.moveActive)
					{
						gAxisCtrl[idxAxis].step = STATE_READY;
					}
				}

				if(gDS1119_Axis[idxAxis].info.status != 0)
				{
					gAxisCtrl[idxAxis].errorID = gDS1119_Axis[idxAxis].info.status;
					strcpy(gAxisCtrl[idxAxis].errorText,gDS1119_Axis[idxAxis].info.errorText);
					gAxisCtrl[idxAxis].step = STATE_ERROR;
				}
				break;

			case STATE_MOVE_JOG_NEG:
				gDS1119_Axis[idxAxis].cmd.velocity = gAxisCtrl[idxAxis].cmd.jogNeg;

				gDS1119_Axis[idxAxis].param.speed  = -gAxisCtrl[idxAxis].param.speed;
				gDS1119_Axis[idxAxis].param.acceleration = gAxisCtrl[idxAxis].param.acceleration;
				gDS1119_Axis[idxAxis].param.deceleration = gAxisCtrl[idxAxis].param.deceleration;

				if(1 == gAxisCtrl[idxAxis].cmd.stop)
				{
					gAxisCtrl[idxAxis].cmd.stop   = 0;
					gAxisCtrl[idxAxis].cmd.jogNeg = 0;
					gDS1119_Axis[idxAxis].cmd.velocity = 0;
					gDS1119_Axis[idxAxis].cmd.stop     = 1;
					gAxisCtrl[idxAxis].step = STATE_STOP;
				}
				else if(0 == gDS1119_Axis[idxAxis].cmd.velocity)
				{
					if(0 == gDS1119_Axis[idxAxis].info.moveActive)
					{
						gAxisCtrl[idxAxis].step = STATE_READY;
					}
				}

				if(gDS1119_Axis[idxAxis].info.status != 0)
				{
					gAxisCtrl[idxAxis].errorID = gDS1119_Axis[idxAxis].info.status;
					strcpy(gAxisCtrl[idxAxis].errorText,gDS1119_Axis[idxAxis].info.errorText);
					gAxisCtrl[idxAxis].step = STATE_ERROR;
				}
				break;

			case STATE_MOVE_ABSOLUTE:
				gDS1119_Axis[idxAxis].param.position = gAxisCtrl[idxAxis].param.position;
				gDS1119_Axis[idxAxis].param.speed    = gAxisCtrl[idxAxis].param.speed;
				gDS1119_Axis[idxAxis].param.acceleration = gAxisCtrl[idxAxis].param.acceleration;
				gDS1119_Axis[idxAxis].param.deceleration = gAxisCtrl[idxAxis].param.deceleration;

				if(1 == gAxisCtrl[idxAxis].cmd.stop)
				{
					gAxisCtrl[idxAxis].cmd.stop = 0;
					gDS1119_Axis[idxAxis].cmd.stop = 1;
					gAxisCtrl[idxAxis].step = STATE_STOP;
				}
				else if(0 == gDS1119_Axis[idxAxis].info.moveActive)
				{
					gAxisCtrl[idxAxis].step = STATE_READY;
				}

				if(gDS1119_Axis[idxAxis].info.status != 0)
				{
					gAxisCtrl[idxAxis].errorID = gDS1119_Axis[idxAxis].info.status;
					strcpy(gAxisCtrl[idxAxis].errorText,gDS1119_Axis[idxAxis].info.errorText);
					gAxisCtrl[idxAxis].step = STATE_ERROR;
				}
				break;

			case STATE_MOVE_RELATIVE:
				gDS1119_Axis[idxAxis].param.position = gAxisCtrl[idxAxis].param.position;
				gDS1119_Axis[idxAxis].param.speed    = gAxisCtrl[idxAxis].param.speed;
				gDS1119_Axis[idxAxis].param.acceleration = gAxisCtrl[idxAxis].param.acceleration;
				gDS1119_Axis[idxAxis].param.deceleration = gAxisCtrl[idxAxis].param.deceleration;

				if(1 == gAxisCtrl[idxAxis].cmd.stop)
				{
					gAxisCtrl[idxAxis].cmd.stop = 0;
					gDS1119_Axis[idxAxis].cmd.stop = 1;
					gAxisCtrl[idxAxis].step = STATE_STOP;
				}
				else if(0 == gDS1119_Axis[idxAxis].info.moveActive)
				{
					gAxisCtrl[idxAxis].step = STATE_READY;
				}

				if(gDS1119_Axis[idxAxis].info.status != 0)
				{
					gAxisCtrl[idxAxis].errorID = gDS1119_Axis[idxAxis].info.status;
					strcpy(gAxisCtrl[idxAxis].errorText,gDS1119_Axis[idxAxis].info.errorText);
					gAxisCtrl[idxAxis].step = STATE_ERROR;
				}
				break;

			case STATE_ERROR:
				if(1 == gAxisCtrl[idxAxis].cmd.acknowledge)
				{
					gAxisCtrl[idxAxis].errorID = 0;
					strcpy(gAxisCtrl[idxAxis].errorText," ");
					gDS1119_Axis[idxAxis].cmd.acknowledge = 1;
					errAckCounter = 0;
					gAxisCtrl[idxAxis].step = STATE_ERROR_RESET;
				}
				break;

			case STATE_ERROR_RESET:
				errAckCounter++;
				if(0 == gDS1119_Axis[idxAxis].info.status)
				{
					gAxisCtrl[idxAxis].step = STATE_WAIT;
				}
				else
				{
					if(errAckCounter > 200)		/* 800 ms */
					{
						gAxisCtrl[idxAxis].step = STATE_WAIT;
															/* error can not acknowledge  */
					}
				}
				break;

		}/* gAxisCtrl[idxAxis].step */

		/* call function DS  */
		DS( &gDS1119_Axis[idxAxis]);

		gAxisCtrl[idxAxis].bReady = ((0 == gAxisCtrl[idxAxis].errorID)        &&
		                             (1 == gDS1119_Axis[idxAxis].info.powerOn)&&
		                             (1 == gDS1119_Axis[idxAxis].info.homingOk));

	}/* for(idxAxis=0;idxAxis<AXIS_NUM_MAX;idxAxis++) */
}/* end of _CYCLIC */
```

#### axisctrl.var
```iecst
VAR
	idxAxis	:UINT;
	errAckCounter	:UINT;
END_VAR
```

### Package Logical/comm - communication with third party equipment

### Program Logical/comm/modem (ANSIC, version 1.00.0) - modem configure / frame drive

#### modem.typ - Local data types
```iecst
(********************************************************************
 * COPYRIGHT --  B&R
 ********************************************************************
 * Program: modem
 * File: modem.typ
 * Author: lij
 * Created: March 06, 2013
 ********************************************************************
 * Local data types of program modem
 ********************************************************************)

TYPE
	BRTransfer : 	STRUCT
		Command : STRING[20];
	END_STRUCT;
END_TYPE
```
